KUKA KRL program: f1_Kuka_APT202T02S02.SRC

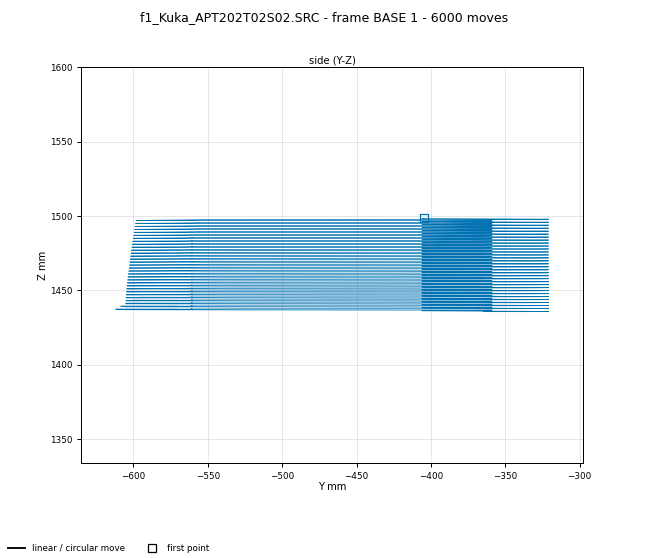
[picture p0: tool path of f1_Kuka_APT202T02S02.SRC in frame BASE 1, 6000 of 6001 moves have a stored position in this frame; points joined in program order, loops and branches not executed]
&ACCESS RVP
&REL 2
&PARAM TEMPLATE = C:\KRC\Roboter\Template\vorgabe
&PARAM EDITMASK = *
DEF f1_Kuka_APT202T02S02()


;FOLD INI;%{PE}%V3.2.0,%MKUKATPBASIS,%CINIT,%VCOMMON,%P
  ;FOLD BAS INI;%{E}%V3.2.0,%MKUKATPBASIS,%CINIT,%VINIT,%P
    GLOBAL INTERRUPT DECL 3 WHEN $STOPMESS==TRUE DO IR_STOPM ( )
    INTERRUPT ON 3
    BAS (#INITMOV,0 )
  ;ENDFOLD (BAS INI)
  ;FOLD USER INI;%{E}%V3.2.0,%MKUKATPUSER,%CINIT,%VINIT,%P
    ;Make your modifications here
  ;ENDFOLD (USER INI)
;ENDFOLD (INI)


;*** Make Null PTP Move
  PTP $pos_act

;*** Auto Load The Correct TOOL Data
  $tool=tool_data[2]

;*** Auto Load The Correct BASE Data
  $base=base_data[1]

  $ADVANCE = 5

;*** Restate Last Velocity
MMPM(30000.0)
SetRPM(8000)
LIN {X -0.079,Y -404.735,Z 1498.391,A 0.000,B 0.000,C 90.000,E1 286.441} C_DIS
LIN {X 0.214,Y -406.099,Z 1498.364,A 0.000,B 0.000,C 90.000,E1 281.535} C_DIS
LIN {X -0.176,Y -406.094,Z 1498.362,A 0.000,B 0.000,C 90.000,E1 281.243} C_DIS
LIN {X -0.097,Y -405.680,Z 1498.333,A 0.000,B 0.000,C 90.000,E1 276.024} C_DIS
LIN {X -0.165,Y -405.058,Z 1498.328,A 0.000,B 0.000,C 90.000,E1 274.992} C_DIS
LIN {X -0.060,Y -403.497,Z 1498.304,A 0.000,B 0.000,C 90.000,E1 270.802} C_DIS
LIN {X -0.092,Y -403.288,Z 1498.302,A 0.000,B 0.000,C 90.000,E1 270.458} C_DIS
LIN {X 0.091,Y -398.931,Z 1498.271,A 0.000,B 0.000,C 90.000,E1 264.837} C_DIS
LIN {X -0.040,Y -393.108,Z 1498.242,A 0.000,B 0.000,C 90.000,E1 259.567} C_DIS
LIN {X -0.079,Y -392.835,Z 1498.240,A 0.000,B 0.000,C 90.000,E1 259.218} C_DIS
LIN {X 0.034,Y -385.993,Z 1498.212,A 0.000,B 0.000,C 90.000,E1 254.212} C_DIS
LIN {X -0.026,Y -385.267,Z 1498.208,A 0.000,B 0.000,C 90.000,E1 253.504} C_DIS
LIN {X -0.004,Y -384.768,Z 1498.206,A 0.000,B 0.000,C 90.000,E1 253.142} C_DIS
LIN {X 0.221,Y -377.973,Z 1498.182,A 0.000,B 0.000,C 90.000,E1 248.773} C_DIS
LIN {X -0.044,Y -376.233,Z 1498.174,A 0.000,B 0.000,C 90.000,E1 247.358} C_DIS
LIN {X 0.057,Y -374.944,Z 1498.170,A 0.000,B 0.000,C 90.000,E1 246.613} C_DIS
LIN {X -0.208,Y -368.417,Z 1498.148,A 0.000,B 0.000,C 90.000,E1 242.615} C_DIS
LIN {X 0.097,Y -366.047,Z 1498.137,A 0.000,B 0.000,C 90.000,E1 240.717} C_DIS
LIN {X 0.004,Y -359.196,Z 1498.115,A 0.000,B 0.000,C 90.000,E1 236.628} C_DIS
LIN {X 0.021,Y -355.842,Z 1498.100,A 0.000,B 0.000,C 90.000,E1 233.989} C_DIS
LIN {X -0.173,Y -348.793,Z 1498.075,A 0.000,B 0.000,C 90.000,E1 229.461} C_DIS
LIN {X -0.097,Y -346.185,Z 1498.062,A 0.000,B 0.000,C 90.000,E1 227.148} C_DIS
LIN {X -0.088,Y -345.065,Z 1498.058,A 0.000,B 0.000,C 90.000,E1 226.377} C_DIS
LIN {X 0.094,Y -338.586,Z 1498.030,A 0.000,B 0.000,C 90.000,E1 221.310} C_DIS
LIN {X 0.094,Y -336.840,Z 1498.019,A 0.000,B 0.000,C 90.000,E1 219.358} C_DIS
LIN {X 0.014,Y -330.861,Z 1497.988,A 0.000,B 0.000,C 90.000,E1 213.865} C_DIS
LIN {X 0.149,Y -329.296,Z 1497.975,A 0.000,B 0.000,C 90.000,E1 211.465} C_DIS
LIN {X -0.154,Y -324.669,Z 1497.942,A 0.000,B 0.000,C 90.000,E1 205.540} C_DIS
LIN {X 0.174,Y -323.837,Z 1497.928,A 0.000,B 0.000,C 90.000,E1 203.078} C_DIS
LIN {X -0.017,Y -321.124,Z 1497.881,A 0.000,B 0.000,C 90.000,E1 194.662} C_DIS
LIN {X 0.138,Y -320.932,Z 1497.877,A 0.000,B 0.000,C 90.000,E1 193.828} C_DIS
LIN {X -0.076,Y -321.562,Z 1497.832,A 0.000,B 0.000,C 90.000,E1 185.796} C_DIS
LIN {X -0.143,Y -324.415,Z 1497.790,A 0.000,B 0.000,C 90.000,E1 178.165} C_DIS
LIN {X -0.141,Y -325.376,Z 1497.783,A 0.000,B 0.000,C 90.000,E1 176.963} C_DIS
LIN {X -0.100,Y -329.112,Z 1497.750,A 0.000,B 0.000,C 90.000,E1 170.971} C_DIS
LIN {X 0.061,Y -334.260,Z 1497.726,A 0.000,B 0.000,C 90.000,E1 166.589} C_DIS
LIN {X 0.067,Y -335.488,Z 1497.719,A 0.000,B 0.000,C 90.000,E1 165.408} C_DIS
LIN {X 0.143,Y -340.932,Z 1497.695,A 0.000,B 0.000,C 90.000,E1 161.094} C_DIS
LIN {X -0.172,Y -342.138,Z 1497.691,A 0.000,B 0.000,C 90.000,E1 160.369} C_DIS
LIN {X -0.058,Y -347.939,Z 1497.667,A 0.000,B 0.000,C 90.000,E1 156.102} C_DIS
LIN {X -0.081,Y -354.259,Z 1497.648,A 0.000,B 0.000,C 90.000,E1 152.666} C_DIS
LIN {X -0.222,Y -361.406,Z 1497.625,A 0.000,B 0.000,C 90.000,E1 148.535} C_DIS
LIN {X 0.128,Y -363.944,Z 1497.618,A 0.000,B 0.000,C 90.000,E1 147.248} C_DIS
LIN {X 0.147,Y -524.568,Z 1497.618,A 0.000,B 0.000,C 90.000,E1 147.248} C_DIS
LIN {X 0.123,Y -527.252,Z 1497.617,A 0.000,B 0.000,C 90.000,E1 147.120} C_DIS
LIN {X 0.098,Y -528.648,Z 1497.617,A 0.000,B 0.000,C 90.000,E1 146.993} C_DIS
LIN {X -0.114,Y -530.734,Z 1497.615,A 0.000,B 0.000,C 90.000,E1 146.755} C_DIS
LIN {X 0.153,Y -533.334,Z 1497.613,A 0.000,B 0.000,C 90.000,E1 146.294} C_DIS
LIN {X 0.143,Y -534.740,Z 1497.611,A 0.000,B 0.000,C 90.000,E1 146.008} C_DIS
LIN {X -0.014,Y -536.490,Z 1497.609,A 0.000,B 0.000,C 90.000,E1 145.595} C_DIS
LIN {X -0.007,Y -538.436,Z 1497.606,A 0.000,B 0.000,C 90.000,E1 145.022} C_DIS
LIN {X -0.295,Y -540.027,Z 1497.603,A 0.000,B 0.000,C 90.000,E1 144.482} C_DIS
LIN {X -0.213,Y -542.835,Z 1497.596,A 0.000,B 0.000,C 90.000,E1 143.336} C_DIS
LIN {X -0.052,Y -545.857,Z 1497.588,A 0.000,B 0.000,C 90.000,E1 141.904} C_DIS
LIN {X 0.073,Y -548.299,Z 1497.581,A 0.000,B 0.000,C 90.000,E1 140.481} C_DIS
LIN {X -0.110,Y -550.441,Z 1497.573,A 0.000,B 0.000,C 90.000,E1 139.094} C_DIS
LIN {X 0.036,Y -551.981,Z 1497.567,A 0.000,B 0.000,C 90.000,E1 137.957} C_DIS
LIN {X -0.256,Y -553.028,Z 1497.562,A 0.000,B 0.000,C 90.000,E1 137.148} C_DIS
LIN {X -0.045,Y -554.642,Z 1497.554,A 0.000,B 0.000,C 90.000,E1 135.729} C_DIS
LIN {X 0.139,Y -555.726,Z 1497.548,A 0.000,B 0.000,C 90.000,E1 134.595} C_DIS
LIN {X -0.006,Y -556.926,Z 1497.540,A 0.000,B 0.000,C 90.000,E1 133.218} C_DIS
LIN {X -0.108,Y -557.910,Z 1497.532,A 0.000,B 0.000,C 90.000,E1 131.838} C_DIS
LIN {X -0.191,Y -558.747,Z 1497.525,A 0.000,B 0.000,C 90.000,E1 130.458} C_DIS
LIN {X 0.161,Y -559.408,Z 1497.517,A 0.000,B 0.000,C 90.000,E1 129.036} C_DIS
LIN {X 0.170,Y -559.997,Z 1497.509,A 0.000,B 0.000,C 90.000,E1 127.649} C_DIS
LIN {X -0.243,Y -560.290,Z 1497.503,A 0.000,B 0.000,C 90.000,E1 126.583} C_DIS
LIN {X -0.099,Y -560.494,Z 1497.495,A 0.000,B 0.000,C 90.000,E1 125.185} C_DIS
LIN {X 0.181,Y -560.465,Z 1497.491,A 0.000,B 0.000,C 90.000,E1 124.326} C_DIS
LIN {X 0.011,Y -560.350,Z 1497.483,A 0.000,B 0.000,C 90.000,E1 122.959} C_DIS
LIN {X 0.188,Y -560.363,Z 1497.472,A 0.000,B 0.000,C 90.000,E1 121.003} C_DIS
LIN {X 0.280,Y -560.586,Z 1497.463,A 0.000,B 0.000,C 90.000,E1 119.333} C_DIS
LIN {X -0.170,Y -560.853,Z 1497.454,A 0.000,B 0.000,C 90.000,E1 117.719} C_DIS
LIN {X 0.244,Y -561.212,Z 1497.442,A 0.000,B 0.000,C 90.000,E1 115.463} C_DIS
LIN {X 0.063,Y -561.585,Z 1497.432,A 0.000,B 0.000,C 90.000,E1 113.823} C_DIS
LIN {X 0.068,Y -561.889,Z 1497.426,A 0.000,B 0.000,C 90.000,E1 112.717} C_DIS
LIN {X -0.004,Y -562.293,Z 1497.416,A 0.000,B 0.000,C 90.000,E1 110.791} C_DIS
LIN {X -0.075,Y -562.700,Z 1497.406,A 0.000,B 0.000,C 90.000,E1 109.141} C_DIS
LIN {X 0.211,Y -563.076,Z 1497.397,A 0.000,B 0.000,C 90.000,E1 107.457} C_DIS
LIN {X -0.196,Y -563.524,Z 1497.388,A 0.000,B 0.000,C 90.000,E1 105.843} C_DIS
LIN {X 0.101,Y -564.102,Z 1497.377,A 0.000,B 0.000,C 90.000,E1 103.883} C_DIS
LIN {X -0.237,Y -564.827,Z 1497.365,A 0.000,B 0.000,C 90.000,E1 101.715} C_DIS
LIN {X 0.046,Y -565.361,Z 1497.357,A 0.000,B 0.000,C 90.000,E1 100.310} C_DIS
LIN {X 0.066,Y -565.901,Z 1497.351,A 0.000,B 0.000,C 90.000,E1 99.208} C_DIS
LIN {X 0.262,Y -566.469,Z 1497.344,A 0.000,B 0.000,C 90.000,E1 97.814} C_DIS
LIN {X -0.210,Y -567.729,Z 1497.330,A 0.000,B 0.000,C 90.000,E1 95.391} C_DIS
LIN {X -0.124,Y -568.501,Z 1497.322,A 0.000,B 0.000,C 90.000,E1 94.012} C_DIS
LIN {X -0.182,Y -569.180,Z 1497.316,A 0.000,B 0.000,C 90.000,E1 92.922} C_DIS
LIN {X -0.104,Y -570.043,Z 1497.309,A 0.000,B 0.000,C 90.000,E1 91.547} C_DIS
LIN {X 0.111,Y -571.078,Z 1497.299,A 0.000,B 0.000,C 90.000,E1 89.885} C_DIS
LIN {X -0.069,Y -572.412,Z 1497.289,A 0.000,B 0.000,C 90.000,E1 87.993} C_DIS
LIN {X 0.076,Y -573.269,Z 1497.281,A 0.000,B 0.000,C 90.000,E1 86.617} C_DIS
LIN {X -0.165,Y -574.340,Z 1497.272,A 0.000,B 0.000,C 90.000,E1 85.008} C_DIS
LIN {X 0.241,Y -575.491,Z 1497.263,A 0.000,B 0.000,C 90.000,E1 83.337} C_DIS
LIN {X -0.065,Y -577.062,Z 1497.251,A 0.000,B 0.000,C 90.000,E1 81.197} C_DIS
LIN {X 0.101,Y -578.510,Z 1497.241,A 0.000,B 0.000,C 90.000,E1 79.285} C_DIS
LIN {X -0.055,Y -580.003,Z 1497.230,A 0.000,B 0.000,C 90.000,E1 77.409} C_DIS
LIN {X 0.301,Y -581.227,Z 1497.221,A 0.000,B 0.000,C 90.000,E1 75.755} C_DIS
LIN {X 0.121,Y -582.355,Z 1497.212,A 0.000,B 0.000,C 90.000,E1 74.157} C_DIS
LIN {X 0.116,Y -583.325,Z 1497.203,A 0.000,B 0.000,C 90.000,E1 72.543} C_DIS
LIN {X -0.097,Y -584.064,Z 1497.196,A 0.000,B 0.000,C 90.000,E1 71.221} C_DIS
LIN {X 0.301,Y -584.970,Z 1497.187,A 0.000,B 0.000,C 90.000,E1 69.571} C_DIS
LIN {X -0.302,Y -586.230,Z 1497.175,A 0.000,B 0.000,C 90.000,E1 67.486} C_DIS
LIN {X -0.310,Y -587.282,Z 1497.164,A 0.000,B 0.000,C 90.000,E1 65.613} C_DIS
LIN {X -0.052,Y -588.468,Z 1497.154,A 0.000,B 0.000,C 90.000,E1 63.717} C_DIS
LIN {X -0.032,Y -589.765,Z 1497.144,A 0.000,B 0.000,C 90.000,E1 61.847} C_DIS
LIN {X -0.108,Y -590.882,Z 1497.135,A 0.000,B 0.000,C 90.000,E1 60.255} C_DIS
LIN {X -0.260,Y -592.270,Z 1497.124,A 0.000,B 0.000,C 90.000,E1 58.408} C_DIS
LIN {X 0.022,Y -593.566,Z 1497.116,A 0.000,B 0.000,C 90.000,E1 56.786} C_DIS
LIN {X -0.056,Y -594.604,Z 1497.108,A 0.000,B 0.000,C 90.000,E1 55.468} C_DIS
LIN {X 0.106,Y -595.700,Z 1497.099,A 0.000,B 0.000,C 90.000,E1 53.863} C_DIS
LIN {X 0.310,Y -596.099,Z 1497.095,A 0.000,B 0.000,C 90.000,E1 53.050} C_DIS
LIN {X -0.227,Y -596.917,Z 1497.085,A 0.000,B 0.000,C 90.000,E1 51.251} C_DIS
LIN {X -0.229,Y -597.429,Z 1497.079,A 0.000,B 0.000,C 90.000,E1 50.194} C_DIS
LIN {X 0.003,Y -597.888,Z 1497.074,A 0.000,B 0.000,C 90.000,E1 49.380} C_DIS
LIN {X 0.014,Y -598.188,Z 1497.068,A 0.000,B 0.000,C 90.000,E1 48.324} C_DIS
LIN {X 0.020,Y -598.255,Z 1497.063,A 0.000,B 0.000,C 90.000,E1 47.268} C_DIS
LIN {X 0.212,Y -598.199,Z 1497.058,A 0.000,B 0.000,C 90.000,E1 46.458} C_DIS
LIN {X -0.024,Y -597.979,Z 1497.051,A 0.000,B 0.000,C 90.000,E1 45.162} C_DIS
LIN {X -0.043,Y -597.462,Z 1497.045,A 0.000,B 0.000,C 90.000,E1 44.109} C_DIS
LIN {X 0.144,Y -596.988,Z 1497.041,A 0.000,B 0.000,C 90.000,E1 43.299} C_DIS
LIN {X -0.090,Y -595.920,Z 1497.033,A 0.000,B 0.000,C 90.000,E1 42.000} C_DIS
LIN {X -0.324,Y -595.174,Z 1497.029,A 0.000,B 0.000,C 90.000,E1 41.229} C_DIS
LIN {X -0.132,Y -593.586,Z 1497.022,A 0.000,B 0.000,C 90.000,E1 39.886} C_DIS
LIN {X 0.062,Y -592.515,Z 1497.017,A 0.000,B 0.000,C 90.000,E1 39.072} C_DIS
LIN {X 0.200,Y -590.340,Z 1497.010,A 0.000,B 0.000,C 90.000,E1 37.729} C_DIS
LIN {X 0.198,Y -588.199,Z 1497.004,A 0.000,B 0.000,C 90.000,E1 36.664} C_DIS
LIN {X -0.025,Y -586.372,Z 1496.999,A 0.000,B 0.000,C 90.000,E1 35.884} C_DIS
LIN {X -0.268,Y -584.413,Z 1496.995,A 0.000,B 0.000,C 90.000,E1 35.105} C_DIS
LIN {X -0.050,Y -582.104,Z 1496.990,A 0.000,B 0.000,C 90.000,E1 34.278} C_DIS
LIN {X -0.175,Y -578.675,Z 1496.984,A 0.000,B 0.000,C 90.000,E1 33.214} C_DIS
LIN {X -0.336,Y -575.589,Z 1496.980,A 0.000,B 0.000,C 90.000,E1 32.418} C_DIS
LIN {X -0.050,Y -573.175,Z 1496.977,A 0.000,B 0.000,C 90.000,E1 31.848} C_DIS
LIN {X -0.304,Y -570.965,Z 1496.975,A 0.000,B 0.000,C 90.000,E1 31.465} C_DIS
LIN {X 0.218,Y -568.308,Z 1496.972,A 0.000,B 0.000,C 90.000,E1 31.003} C_DIS
LIN {X 0.039,Y -566.164,Z 1496.971,A 0.000,B 0.000,C 90.000,E1 30.747} C_DIS
LIN {X 0.235,Y -564.885,Z 1496.970,A 0.000,B 0.000,C 90.000,E1 30.590} C_DIS
LIN {X 0.084,Y -562.667,Z 1496.969,A 0.000,B 0.000,C 90.000,E1 30.413} C_DIS
LIN {X -0.176,Y -560.913,Z 1496.969,A 0.000,B 0.000,C 90.000,E1 30.335} C_DIS
LIN {X 0.114,Y -559.281,Z 1496.968,A 0.000,B 0.000,C 90.000,E1 30.256} C_DIS
LIN {X 0.055,Y -390.789,Z 1496.968,A 0.000,B 0.000,C 90.000,E1 30.256} C_DIS
LIN {X -0.100,Y -383.744,Z 1496.942,A 0.000,B 0.000,C 90.000,E1 25.591} C_DIS
LIN {X 0.062,Y -382.915,Z 1496.938,A 0.000,B 0.000,C 90.000,E1 24.847} C_DIS
LIN {X 0.168,Y -376.206,Z 1496.912,A 0.000,B 0.000,C 90.000,E1 20.120} C_DIS
LIN {X 0.036,Y -373.711,Z 1496.898,A 0.000,B 0.000,C 90.000,E1 17.583} C_DIS
LIN {X 0.172,Y -368.106,Z 1496.869,A 0.000,B 0.000,C 90.000,E1 12.411} C_DIS
LIN {X -0.022,Y -366.430,Z 1496.855,A 0.000,B 0.000,C 90.000,E1 9.849} C_DIS
LIN {X -0.084,Y -361.753,Z 1496.822,A 0.000,B 0.000,C 90.000,E1 3.898} C_DIS
LIN {X 0.163,Y -360.877,Z 1496.801,A 0.000,B 0.000,C 90.000,E1 0.115} C_DIS
LIN {X -0.053,Y -359.426,Z 1496.770,A 0.000,B 0.000,C 90.000,E1 354.546} C_DIS
LIN {X 0.070,Y -358.890,Z 1496.759,A 0.000,B 0.000,C 90.000,E1 352.648} C_DIS
LIN {X -0.020,Y -359.563,Z 1496.726,A 0.000,B 0.000,C 90.000,E1 346.645} C_DIS
LIN {X 0.001,Y -361.801,Z 1496.684,A 0.000,B 0.000,C 90.000,E1 339.135} C_DIS
LIN {X -0.154,Y -362.053,Z 1496.680,A 0.000,B 0.000,C 90.000,E1 338.411} C_DIS
LIN {X 0.189,Y -365.980,Z 1496.643,A 0.000,B 0.000,C 90.000,E1 331.641} C_DIS
LIN {X 0.029,Y -366.387,Z 1496.639,A 0.000,B 0.000,C 90.000,E1 330.923} C_DIS
LIN {X -0.031,Y -371.355,Z 1496.604,A 0.000,B 0.000,C 90.000,E1 324.642} C_DIS
LIN {X -0.043,Y -371.766,Z 1496.602,A 0.000,B 0.000,C 90.000,E1 324.276} C_DIS
LIN {X 0.013,Y -377.358,Z 1496.567,A 0.000,B 0.000,C 90.000,E1 318.038} C_DIS
LIN {X 0.012,Y -378.235,Z 1496.563,A 0.000,B 0.000,C 90.000,E1 317.310} C_DIS
LIN {X 0.002,Y -383.940,Z 1496.531,A 0.000,B 0.000,C 90.000,E1 311.515} C_DIS
LIN {X 0.088,Y -384.893,Z 1496.527,A 0.000,B 0.000,C 90.000,E1 310.782} C_DIS
LIN {X 0.262,Y -390.610,Z 1496.495,A 0.000,B 0.000,C 90.000,E1 305.025} C_DIS
LIN {X 0.106,Y -391.104,Z 1496.493,A 0.000,B 0.000,C 90.000,E1 304.692} C_DIS
LIN {X 0.022,Y -391.648,Z 1496.489,A 0.000,B 0.000,C 90.000,E1 303.992} C_DIS
LIN {X -0.080,Y -396.825,Z 1496.459,A 0.000,B 0.000,C 90.000,E1 298.693} C_DIS
LIN {X -0.210,Y -397.120,Z 1496.457,A 0.000,B 0.000,C 90.000,E1 298.359} C_DIS
LIN {X -0.055,Y -401.597,Z 1496.426,A 0.000,B 0.000,C 90.000,E1 292.717} C_DIS
LIN {X 0.222,Y -404.659,Z 1496.395,A 0.000,B 0.000,C 90.000,E1 287.094} C_DIS
LIN {X -0.079,Y -404.735,Z 1496.391,A 0.000,B 0.000,C 90.000,E1 286.441} C_DIS
LIN {X 0.214,Y -406.099,Z 1496.364,A 0.000,B 0.000,C 90.000,E1 281.535} C_DIS
LIN {X -0.176,Y -406.094,Z 1496.362,A 0.000,B 0.000,C 90.000,E1 281.243} C_DIS
LIN {X -0.097,Y -405.680,Z 1496.333,A 0.000,B 0.000,C 90.000,E1 276.024} C_DIS
LIN {X -0.165,Y -405.058,Z 1496.328,A 0.000,B 0.000,C 90.000,E1 274.992} C_DIS
LIN {X -0.060,Y -403.497,Z 1496.304,A 0.000,B 0.000,C 90.000,E1 270.802} C_DIS
LIN {X -0.092,Y -403.288,Z 1496.302,A 0.000,B 0.000,C 90.000,E1 270.458} C_DIS
LIN {X 0.091,Y -398.931,Z 1496.271,A 0.000,B 0.000,C 90.000,E1 264.837} C_DIS
LIN {X -0.040,Y -393.108,Z 1496.242,A 0.000,B 0.000,C 90.000,E1 259.567} C_DIS
LIN {X -0.079,Y -392.835,Z 1496.240,A 0.000,B 0.000,C 90.000,E1 259.218} C_DIS
LIN {X 0.034,Y -385.993,Z 1496.212,A 0.000,B 0.000,C 90.000,E1 254.212} C_DIS
LIN {X -0.026,Y -385.267,Z 1496.208,A 0.000,B 0.000,C 90.000,E1 253.504} C_DIS
LIN {X -0.004,Y -384.768,Z 1496.206,A 0.000,B 0.000,C 90.000,E1 253.142} C_DIS
LIN {X 0.221,Y -377.973,Z 1496.182,A 0.000,B 0.000,C 90.000,E1 248.773} C_DIS
LIN {X -0.044,Y -376.233,Z 1496.174,A 0.000,B 0.000,C 90.000,E1 247.358} C_DIS
LIN {X 0.057,Y -374.944,Z 1496.170,A 0.000,B 0.000,C 90.000,E1 246.613} C_DIS
LIN {X -0.208,Y -368.417,Z 1496.148,A 0.000,B 0.000,C 90.000,E1 242.615} C_DIS
LIN {X 0.097,Y -366.047,Z 1496.137,A 0.000,B 0.000,C 90.000,E1 240.717} C_DIS
LIN {X 0.004,Y -359.196,Z 1496.115,A 0.000,B 0.000,C 90.000,E1 236.628} C_DIS
LIN {X 0.021,Y -355.842,Z 1496.100,A 0.000,B 0.000,C 90.000,E1 233.989} C_DIS
LIN {X -0.173,Y -348.793,Z 1496.075,A 0.000,B 0.000,C 90.000,E1 229.461} C_DIS
LIN {X -0.097,Y -346.185,Z 1496.062,A 0.000,B 0.000,C 90.000,E1 227.148} C_DIS
LIN {X -0.088,Y -345.065,Z 1496.058,A 0.000,B 0.000,C 90.000,E1 226.377} C_DIS
LIN {X 0.094,Y -338.586,Z 1496.030,A 0.000,B 0.000,C 90.000,E1 221.310} C_DIS
LIN {X 0.094,Y -336.840,Z 1496.019,A 0.000,B 0.000,C 90.000,E1 219.358} C_DIS
LIN {X 0.014,Y -330.861,Z 1495.988,A 0.000,B 0.000,C 90.000,E1 213.865} C_DIS
LIN {X 0.149,Y -329.296,Z 1495.975,A 0.000,B 0.000,C 90.000,E1 211.465} C_DIS
LIN {X -0.154,Y -324.669,Z 1495.942,A 0.000,B 0.000,C 90.000,E1 205.540} C_DIS
LIN {X 0.174,Y -323.837,Z 1495.928,A 0.000,B 0.000,C 90.000,E1 203.078} C_DIS
LIN {X -0.017,Y -321.124,Z 1495.881,A 0.000,B 0.000,C 90.000,E1 194.662} C_DIS
LIN {X 0.138,Y -320.932,Z 1495.877,A 0.000,B 0.000,C 90.000,E1 193.828} C_DIS
LIN {X -0.076,Y -321.562,Z 1495.832,A 0.000,B 0.000,C 90.000,E1 185.796} C_DIS
LIN {X -0.143,Y -324.415,Z 1495.790,A 0.000,B 0.000,C 90.000,E1 178.165} C_DIS
LIN {X -0.141,Y -325.376,Z 1495.783,A 0.000,B 0.000,C 90.000,E1 176.963} C_DIS
LIN {X -0.100,Y -329.112,Z 1495.750,A 0.000,B 0.000,C 90.000,E1 170.971} C_DIS
LIN {X 0.061,Y -334.260,Z 1495.726,A 0.000,B 0.000,C 90.000,E1 166.589} C_DIS
LIN {X 0.067,Y -335.488,Z 1495.719,A 0.000,B 0.000,C 90.000,E1 165.408} C_DIS
LIN {X 0.143,Y -340.932,Z 1495.695,A 0.000,B 0.000,C 90.000,E1 161.094} C_DIS
LIN {X -0.172,Y -342.138,Z 1495.691,A 0.000,B 0.000,C 90.000,E1 160.369} C_DIS
LIN {X -0.058,Y -347.939,Z 1495.667,A 0.000,B 0.000,C 90.000,E1 156.102} C_DIS
LIN {X -0.081,Y -354.259,Z 1495.648,A 0.000,B 0.000,C 90.000,E1 152.666} C_DIS
LIN {X -0.222,Y -361.406,Z 1495.625,A 0.000,B 0.000,C 90.000,E1 148.535} C_DIS
LIN {X -0.211,Y -362.490,Z 1495.622,A 0.000,B 0.000,C 90.000,E1 147.995} C_DIS
LIN {X 0.110,Y -522.437,Z 1495.622,A 0.000,B 0.000,C 90.000,E1 147.946} C_DIS
LIN {X -0.131,Y -524.949,Z 1495.621,A 0.000,B 0.000,C 90.000,E1 147.867} C_DIS
LIN {X 0.102,Y -526.192,Z 1495.621,A 0.000,B 0.000,C 90.000,E1 147.740} C_DIS
LIN {X 0.059,Y -528.355,Z 1495.620,A 0.000,B 0.000,C 90.000,E1 147.502} C_DIS
LIN {X -0.243,Y -530.287,Z 1495.618,A 0.000,B 0.000,C 90.000,E1 147.248} C_DIS
LIN {X 0.022,Y -532.672,Z 1495.616,A 0.000,B 0.000,C 90.000,E1 146.786} C_DIS
LIN {X -0.147,Y -534.604,Z 1495.613,A 0.000,B 0.000,C 90.000,E1 146.373} C_DIS
LIN {X -0.154,Y -535.744,Z 1495.612,A 0.000,B 0.000,C 90.000,E1 146.087} C_DIS
LIN {X -0.156,Y -537.582,Z 1495.608,A 0.000,B 0.000,C 90.000,E1 145.515} C_DIS
LIN {X 0.003,Y -539.990,Z 1495.604,A 0.000,B 0.000,C 90.000,E1 144.642} C_DIS
LIN {X 0.057,Y -542.139,Z 1495.599,A 0.000,B 0.000,C 90.000,E1 143.783} C_DIS
LIN {X 0.137,Y -544.076,Z 1495.594,A 0.000,B 0.000,C 90.000,E1 142.924} C_DIS
LIN {X -0.192,Y -545.882,Z 1495.589,A 0.000,B 0.000,C 90.000,E1 142.110} C_DIS
LIN {X -0.029,Y -547.881,Z 1495.583,A 0.000,B 0.000,C 90.000,E1 140.964} C_DIS
LIN {X 0.082,Y -549.671,Z 1495.577,A 0.000,B 0.000,C 90.000,E1 139.828} C_DIS
LIN {X 0.224,Y -551.300,Z 1495.571,A 0.000,B 0.000,C 90.000,E1 138.690} C_DIS
LIN {X -0.021,Y -552.782,Z 1495.564,A 0.000,B 0.000,C 90.000,E1 137.595} C_DIS
LIN {X 0.244,Y -554.722,Z 1495.555,A 0.000,B 0.000,C 90.000,E1 135.891} C_DIS
LIN {X 0.035,Y -555.819,Z 1495.549,A 0.000,B 0.000,C 90.000,E1 134.798} C_DIS
LIN {X -0.095,Y -557.046,Z 1495.541,A 0.000,B 0.000,C 90.000,E1 133.419} C_DIS
LIN {X 0.189,Y -558.017,Z 1495.533,A 0.000,B 0.000,C 90.000,E1 132.000} C_DIS
LIN {X 0.030,Y -558.685,Z 1495.527,A 0.000,B 0.000,C 90.000,E1 130.906} C_DIS
LIN {X -0.062,Y -559.255,Z 1495.521,A 0.000,B 0.000,C 90.000,E1 129.806} C_DIS
LIN {X 0.302,Y -559.823,Z 1495.513,A 0.000,B 0.000,C 90.000,E1 128.382} C_DIS
LIN {X -0.208,Y -560.128,Z 1495.509,A 0.000,B 0.000,C 90.000,E1 127.604} C_DIS
LIN {X 0.076,Y -560.338,Z 1495.504,A 0.000,B 0.000,C 90.000,E1 126.744} C_DIS
LIN {X -0.232,Y -560.549,Z 1495.497,A 0.000,B 0.000,C 90.000,E1 125.391} C_DIS
LIN {X -0.174,Y -560.489,Z 1495.490,A 0.000,B 0.000,C 90.000,E1 124.278} C_DIS
LIN {X -0.032,Y -560.362,Z 1495.483,A 0.000,B 0.000,C 90.000,E1 122.880} C_DIS
LIN {X 0.139,Y -560.395,Z 1495.472,A 0.000,B 0.000,C 90.000,E1 120.924} C_DIS
LIN {X -0.047,Y -560.625,Z 1495.463,A 0.000,B 0.000,C 90.000,E1 119.283} C_DIS
LIN {X 0.068,Y -560.940,Z 1495.452,A 0.000,B 0.000,C 90.000,E1 117.334} C_DIS
LIN {X -0.265,Y -561.309,Z 1495.440,A 0.000,B 0.000,C 90.000,E1 115.155} C_DIS
LIN {X -0.126,Y -561.830,Z 1495.429,A 0.000,B 0.000,C 90.000,E1 113.206} C_DIS
LIN {X 0.003,Y -562.154,Z 1495.420,A 0.000,B 0.000,C 90.000,E1 111.535} C_DIS
LIN {X -0.062,Y -562.534,Z 1495.411,A 0.000,B 0.000,C 90.000,E1 109.885} C_DIS
LIN {X -0.126,Y -562.961,Z 1495.401,A 0.000,B 0.000,C 90.000,E1 108.236} C_DIS
LIN {X -0.228,Y -563.464,Z 1495.391,A 0.000,B 0.000,C 90.000,E1 106.315} C_DIS
LIN {X 0.224,Y -564.103,Z 1495.378,A 0.000,B 0.000,C 90.000,E1 104.064} C_DIS
LIN {X 0.232,Y -564.617,Z 1495.369,A 0.000,B 0.000,C 90.000,E1 102.411} C_DIS
LIN {X 0.013,Y -565.272,Z 1495.360,A 0.000,B 0.000,C 90.000,E1 100.782} C_DIS
LIN {X -0.182,Y -566.027,Z 1495.351,A 0.000,B 0.000,C 90.000,E1 99.151} C_DIS
LIN {X 0.018,Y -566.588,Z 1495.343,A 0.000,B 0.000,C 90.000,E1 97.757} C_DIS
LIN {X -0.045,Y -567.731,Z 1495.331,A 0.000,B 0.000,C 90.000,E1 95.568} C_DIS
LIN {X 0.209,Y -568.649,Z 1495.322,A 0.000,B 0.000,C 90.000,E1 93.898} C_DIS
LIN {X 0.154,Y -569.353,Z 1495.316,A 0.000,B 0.000,C 90.000,E1 92.808} C_DIS
LIN {X 0.237,Y -570.216,Z 1495.308,A 0.000,B 0.000,C 90.000,E1 91.432} C_DIS
LIN {X -0.247,Y -571.113,Z 1495.301,A 0.000,B 0.000,C 90.000,E1 90.115} C_DIS
LIN {X -0.009,Y -572.252,Z 1495.292,A 0.000,B 0.000,C 90.000,E1 88.453} C_DIS
LIN {X 0.124,Y -573.175,Z 1495.284,A 0.000,B 0.000,C 90.000,E1 87.078} C_DIS
LIN {X -0.125,Y -574.223,Z 1495.275,A 0.000,B 0.000,C 90.000,E1 85.469} C_DIS
LIN {X 0.273,Y -575.363,Z 1495.266,A 0.000,B 0.000,C 90.000,E1 83.799} C_DIS
LIN {X -0.245,Y -576.726,Z 1495.255,A 0.000,B 0.000,C 90.000,E1 81.951} C_DIS
LIN {X -0.295,Y -577.948,Z 1495.246,A 0.000,B 0.000,C 90.000,E1 80.330} C_DIS
LIN {X 0.006,Y -578.821,Z 1495.240,A 0.000,B 0.000,C 90.000,E1 79.218} C_DIS
LIN {X 0.088,Y -580.090,Z 1495.231,A 0.000,B 0.000,C 90.000,E1 77.589} C_DIS
LIN {X 0.214,Y -581.171,Z 1495.224,A 0.000,B 0.000,C 90.000,E1 76.228} C_DIS
LIN {X -0.192,Y -582.130,Z 1495.216,A 0.000,B 0.000,C 90.000,E1 74.921} C_DIS
LIN {X -0.022,Y -583.002,Z 1495.209,A 0.000,B 0.000,C 90.000,E1 73.559} C_DIS
LIN {X -0.236,Y -583.767,Z 1495.201,A 0.000,B 0.000,C 90.000,E1 72.236} C_DIS
LIN {X -0.101,Y -584.374,Z 1495.195,A 0.000,B 0.000,C 90.000,E1 71.148} C_DIS
LIN {X 0.109,Y -585.258,Z 1495.186,A 0.000,B 0.000,C 90.000,E1 69.518} C_DIS
LIN {X 0.272,Y -586.506,Z 1495.174,A 0.000,B 0.000,C 90.000,E1 67.358} C_DIS
LIN {X 0.274,Y -587.593,Z 1495.164,A 0.000,B 0.000,C 90.000,E1 65.485} C_DIS
LIN {X 0.015,Y -588.761,Z 1495.154,A 0.000,B 0.000,C 90.000,E1 63.640} C_DIS
LIN {X 0.050,Y -590.034,Z 1495.143,A 0.000,B 0.000,C 90.000,E1 61.769} C_DIS
LIN {X -0.307,Y -591.165,Z 1495.134,A 0.000,B 0.000,C 90.000,E1 60.205} C_DIS
LIN {X -0.152,Y -592.596,Z 1495.124,A 0.000,B 0.000,C 90.000,E1 58.329} C_DIS
LIN {X 0.142,Y -593.861,Z 1495.115,A 0.000,B 0.000,C 90.000,E1 56.707} C_DIS
LIN {X 0.074,Y -594.943,Z 1495.108,A 0.000,B 0.000,C 90.000,E1 55.388} C_DIS
LIN {X 0.247,Y -596.049,Z 1495.099,A 0.000,B 0.000,C 90.000,E1 53.783} C_DIS
LIN {X -0.148,Y -596.553,Z 1495.093,A 0.000,B 0.000,C 90.000,E1 52.763} C_DIS
LIN {X -0.067,Y -597.271,Z 1495.084,A 0.000,B 0.000,C 90.000,E1 51.170} C_DIS
LIN {X -0.064,Y -597.787,Z 1495.078,A 0.000,B 0.000,C 90.000,E1 50.114} C_DIS
LIN {X 0.174,Y -598.232,Z 1495.074,A 0.000,B 0.000,C 90.000,E1 49.299} C_DIS
LIN {X 0.190,Y -598.511,Z 1495.068,A 0.000,B 0.000,C 90.000,E1 48.243} C_DIS
LIN {X -0.237,Y -598.581,Z 1495.062,A 0.000,B 0.000,C 90.000,E1 47.229} C_DIS
LIN {X -0.036,Y -598.513,Z 1495.058,A 0.000,B 0.000,C 90.000,E1 46.419} C_DIS
LIN {X 0.168,Y -598.285,Z 1495.051,A 0.000,B 0.000,C 90.000,E1 45.081} C_DIS
LIN {X 0.153,Y -597.773,Z 1495.045,A 0.000,B 0.000,C 90.000,E1 44.028} C_DIS
LIN {X -0.067,Y -597.302,Z 1495.040,A 0.000,B 0.000,C 90.000,E1 43.257} C_DIS
LIN {X 0.113,Y -596.230,Z 1495.033,A 0.000,B 0.000,C 90.000,E1 41.919} C_DIS
LIN {X -0.120,Y -595.446,Z 1495.029,A 0.000,B 0.000,C 90.000,E1 41.148} C_DIS
LIN {X -0.144,Y -594.237,Z 1495.023,A 0.000,B 0.000,C 90.000,E1 40.092} C_DIS
LIN {X -0.189,Y -592.764,Z 1495.017,A 0.000,B 0.000,C 90.000,E1 39.036} C_DIS
LIN {X -0.162,Y -591.058,Z 1495.011,A 0.000,B 0.000,C 90.000,E1 37.971} C_DIS
LIN {X 0.206,Y -589.018,Z 1495.005,A 0.000,B 0.000,C 90.000,E1 36.870} C_DIS
LIN {X -0.211,Y -587.928,Z 1495.002,A 0.000,B 0.000,C 90.000,E1 36.377} C_DIS
LIN {X -0.245,Y -585.364,Z 1494.996,A 0.000,B 0.000,C 90.000,E1 35.311} C_DIS
LIN {X -0.017,Y -583.180,Z 1494.992,A 0.000,B 0.000,C 90.000,E1 34.485} C_DIS
LIN {X -0.127,Y -579.850,Z 1494.986,A 0.000,B 0.000,C 90.000,E1 33.420} C_DIS
LIN {X -0.121,Y -577.955,Z 1494.983,A 0.000,B 0.000,C 90.000,E1 32.880} C_DIS
LIN {X 0.021,Y -574.761,Z 1494.978,A 0.000,B 0.000,C 90.000,E1 32.054} C_DIS
LIN {X -0.091,Y -571.728,Z 1494.974,A 0.000,B 0.000,C 90.000,E1 31.386} C_DIS
LIN {X -0.143,Y -568.756,Z 1494.971,A 0.000,B 0.000,C 90.000,E1 30.846} C_DIS
LIN {X 0.077,Y -565.975,Z 1494.969,A 0.000,B 0.000,C 90.000,E1 30.413} C_DIS
LIN {X 0.178,Y -563.742,Z 1494.968,A 0.000,B 0.000,C 90.000,E1 30.129} C_DIS
LIN {X 0.081,Y -562.439,Z 1494.967,A 0.000,B 0.000,C 90.000,E1 30.001} C_DIS
LIN {X -0.016,Y -559.895,Z 1494.966,A 0.000,B 0.000,C 90.000,E1 29.795} C_DIS
LIN {X 0.159,Y -557.890,Z 1494.965,A 0.000,B 0.000,C 90.000,E1 29.667} C_DIS
LIN {X -0.147,Y -556.512,Z 1494.965,A 0.000,B 0.000,C 90.000,E1 29.667} C_DIS
LIN {X -0.127,Y -389.695,Z 1494.965,A 0.000,B 0.000,C 90.000,E1 29.667} C_DIS
LIN {X 0.087,Y -383.035,Z 1494.939,A 0.000,B 0.000,C 90.000,E1 24.951} C_DIS
LIN {X -0.105,Y -381.915,Z 1494.935,A 0.000,B 0.000,C 90.000,E1 24.259} C_DIS
LIN {X 0.018,Y -375.527,Z 1494.909,A 0.000,B 0.000,C 90.000,E1 19.523} C_DIS
LIN {X 0.012,Y -373.428,Z 1494.896,A 0.000,B 0.000,C 90.000,E1 17.330} C_DIS
LIN {X -0.054,Y -367.906,Z 1494.868,A 0.000,B 0.000,C 90.000,E1 12.187} C_DIS
LIN {X -0.034,Y -366.504,Z 1494.855,A 0.000,B 0.000,C 90.000,E1 9.962} C_DIS
LIN {X -0.099,Y -361.803,Z 1494.822,A 0.000,B 0.000,C 90.000,E1 4.012} C_DIS
LIN {X 0.147,Y -360.903,Z 1494.802,A 0.000,B 0.000,C 90.000,E1 0.229} C_DIS
LIN {X -0.053,Y -359.426,Z 1494.770,A 0.000,B 0.000,C 90.000,E1 354.546} C_DIS
LIN {X 0.070,Y -358.890,Z 1494.759,A 0.000,B 0.000,C 90.000,E1 352.648} C_DIS
LIN {X -0.020,Y -359.563,Z 1494.726,A 0.000,B 0.000,C 90.000,E1 346.645} C_DIS
LIN {X 0.001,Y -361.801,Z 1494.684,A 0.000,B 0.000,C 90.000,E1 339.135} C_DIS
LIN {X -0.154,Y -362.053,Z 1494.680,A 0.000,B 0.000,C 90.000,E1 338.411} C_DIS
LIN {X 0.189,Y -365.980,Z 1494.643,A 0.000,B 0.000,C 90.000,E1 331.641} C_DIS
LIN {X 0.029,Y -366.387,Z 1494.639,A 0.000,B 0.000,C 90.000,E1 330.923} C_DIS
LIN {X -0.031,Y -371.355,Z 1494.604,A 0.000,B 0.000,C 90.000,E1 324.642} C_DIS
LIN {X -0.043,Y -371.766,Z 1494.602,A 0.000,B 0.000,C 90.000,E1 324.276} C_DIS
LIN {X 0.013,Y -377.358,Z 1494.567,A 0.000,B 0.000,C 90.000,E1 318.038} C_DIS
LIN {X 0.012,Y -378.235,Z 1494.563,A 0.000,B 0.000,C 90.000,E1 317.310} C_DIS
LIN {X 0.002,Y -383.940,Z 1494.531,A 0.000,B 0.000,C 90.000,E1 311.515} C_DIS
LIN {X 0.088,Y -384.893,Z 1494.527,A 0.000,B 0.000,C 90.000,E1 310.782} C_DIS
LIN {X 0.262,Y -390.610,Z 1494.495,A 0.000,B 0.000,C 90.000,E1 305.025} C_DIS
LIN {X 0.106,Y -391.104,Z 1494.493,A 0.000,B 0.000,C 90.000,E1 304.692} C_DIS
LIN {X 0.022,Y -391.648,Z 1494.489,A 0.000,B 0.000,C 90.000,E1 303.992} C_DIS
LIN {X -0.080,Y -396.825,Z 1494.459,A 0.000,B 0.000,C 90.000,E1 298.693} C_DIS
LIN {X -0.210,Y -397.120,Z 1494.457,A 0.000,B 0.000,C 90.000,E1 298.359} C_DIS
LIN {X -0.055,Y -401.597,Z 1494.426,A 0.000,B 0.000,C 90.000,E1 292.717} C_DIS
LIN {X 0.222,Y -404.659,Z 1494.395,A 0.000,B 0.000,C 90.000,E1 287.094} C_DIS
LIN {X -0.079,Y -404.735,Z 1494.391,A 0.000,B 0.000,C 90.000,E1 286.441} C_DIS
LIN {X 0.214,Y -406.099,Z 1494.364,A 0.000,B 0.000,C 90.000,E1 281.535} C_DIS
LIN {X -0.176,Y -406.094,Z 1494.362,A 0.000,B 0.000,C 90.000,E1 281.243} C_DIS
LIN {X -0.097,Y -405.680,Z 1494.333,A 0.000,B 0.000,C 90.000,E1 276.024} C_DIS
LIN {X -0.165,Y -405.058,Z 1494.328,A 0.000,B 0.000,C 90.000,E1 274.992} C_DIS
LIN {X -0.060,Y -403.497,Z 1494.304,A 0.000,B 0.000,C 90.000,E1 270.802} C_DIS
LIN {X -0.092,Y -403.288,Z 1494.302,A 0.000,B 0.000,C 90.000,E1 270.458} C_DIS
LIN {X 0.091,Y -398.931,Z 1494.271,A 0.000,B 0.000,C 90.000,E1 264.837} C_DIS
LIN {X -0.040,Y -393.108,Z 1494.242,A 0.000,B 0.000,C 90.000,E1 259.567} C_DIS
LIN {X -0.079,Y -392.835,Z 1494.240,A 0.000,B 0.000,C 90.000,E1 259.218} C_DIS
LIN {X 0.034,Y -385.993,Z 1494.212,A 0.000,B 0.000,C 90.000,E1 254.212} C_DIS
LIN {X -0.026,Y -385.267,Z 1494.208,A 0.000,B 0.000,C 90.000,E1 253.504} C_DIS
LIN {X -0.004,Y -384.768,Z 1494.206,A 0.000,B 0.000,C 90.000,E1 253.142} C_DIS
LIN {X 0.221,Y -377.973,Z 1494.182,A 0.000,B 0.000,C 90.000,E1 248.773} C_DIS
LIN {X -0.044,Y -376.233,Z 1494.174,A 0.000,B 0.000,C 90.000,E1 247.358} C_DIS
LIN {X 0.057,Y -374.944,Z 1494.170,A 0.000,B 0.000,C 90.000,E1 246.613} C_DIS
LIN {X -0.208,Y -368.417,Z 1494.148,A 0.000,B 0.000,C 90.000,E1 242.615} C_DIS
LIN {X 0.097,Y -366.047,Z 1494.137,A 0.000,B 0.000,C 90.000,E1 240.717} C_DIS
LIN {X 0.004,Y -359.196,Z 1494.115,A 0.000,B 0.000,C 90.000,E1 236.628} C_DIS
LIN {X 0.021,Y -355.842,Z 1494.100,A 0.000,B 0.000,C 90.000,E1 233.989} C_DIS
LIN {X -0.173,Y -348.793,Z 1494.075,A 0.000,B 0.000,C 90.000,E1 229.461} C_DIS
LIN {X -0.097,Y -346.185,Z 1494.062,A 0.000,B 0.000,C 90.000,E1 227.148} C_DIS
LIN {X -0.088,Y -345.065,Z 1494.058,A 0.000,B 0.000,C 90.000,E1 226.377} C_DIS
LIN {X 0.094,Y -338.586,Z 1494.030,A 0.000,B 0.000,C 90.000,E1 221.310} C_DIS
LIN {X 0.094,Y -336.840,Z 1494.019,A 0.000,B 0.000,C 90.000,E1 219.358} C_DIS
LIN {X 0.014,Y -330.861,Z 1493.988,A 0.000,B 0.000,C 90.000,E1 213.865} C_DIS
LIN {X 0.149,Y -329.296,Z 1493.975,A 0.000,B 0.000,C 90.000,E1 211.465} C_DIS
LIN {X -0.154,Y -324.669,Z 1493.942,A 0.000,B 0.000,C 90.000,E1 205.540} C_DIS
LIN {X 0.174,Y -323.837,Z 1493.928,A 0.000,B 0.000,C 90.000,E1 203.078} C_DIS
LIN {X -0.017,Y -321.124,Z 1493.881,A 0.000,B 0.000,C 90.000,E1 194.662} C_DIS
LIN {X 0.138,Y -320.932,Z 1493.877,A 0.000,B 0.000,C 90.000,E1 193.828} C_DIS
LIN {X -0.076,Y -321.562,Z 1493.832,A 0.000,B 0.000,C 90.000,E1 185.796} C_DIS
LIN {X -0.143,Y -324.415,Z 1493.790,A 0.000,B 0.000,C 90.000,E1 178.165} C_DIS
LIN {X -0.141,Y -325.376,Z 1493.783,A 0.000,B 0.000,C 90.000,E1 176.963} C_DIS
LIN {X -0.100,Y -329.112,Z 1493.750,A 0.000,B 0.000,C 90.000,E1 170.971} C_DIS
LIN {X 0.061,Y -334.260,Z 1493.726,A 0.000,B 0.000,C 90.000,E1 166.589} C_DIS
LIN {X 0.067,Y -335.488,Z 1493.719,A 0.000,B 0.000,C 90.000,E1 165.408} C_DIS
LIN {X 0.143,Y -340.932,Z 1493.695,A 0.000,B 0.000,C 90.000,E1 161.094} C_DIS
LIN {X -0.172,Y -342.138,Z 1493.691,A 0.000,B 0.000,C 90.000,E1 160.369} C_DIS
LIN {X -0.058,Y -347.939,Z 1493.667,A 0.000,B 0.000,C 90.000,E1 156.102} C_DIS
LIN {X -0.081,Y -354.259,Z 1493.648,A 0.000,B 0.000,C 90.000,E1 152.666} C_DIS
LIN {X -0.124,Y -361.124,Z 1493.626,A 0.000,B 0.000,C 90.000,E1 148.663} C_DIS
LIN {X -0.226,Y -520.265,Z 1493.626,A 0.000,B 0.000,C 90.000,E1 148.663} C_DIS
LIN {X -0.321,Y -523.251,Z 1493.625,A 0.000,B 0.000,C 90.000,E1 148.535} C_DIS
LIN {X 0.132,Y -525.006,Z 1493.624,A 0.000,B 0.000,C 90.000,E1 148.329} C_DIS
LIN {X 0.129,Y -527.116,Z 1493.623,A 0.000,B 0.000,C 90.000,E1 148.074} C_DIS
LIN {X -0.072,Y -529.886,Z 1493.620,A 0.000,B 0.000,C 90.000,E1 147.661} C_DIS
LIN {X -0.256,Y -532.039,Z 1493.618,A 0.000,B 0.000,C 90.000,E1 147.248} C_DIS
LIN {X 0.173,Y -533.297,Z 1493.616,A 0.000,B 0.000,C 90.000,E1 146.914} C_DIS
LIN {X -0.144,Y -535.428,Z 1493.613,A 0.000,B 0.000,C 90.000,E1 146.373} C_DIS
LIN {X -0.150,Y -537.214,Z 1493.610,A 0.000,B 0.000,C 90.000,E1 145.801} C_DIS
LIN {X 0.018,Y -540.443,Z 1493.604,A 0.000,B 0.000,C 90.000,E1 144.642} C_DIS
LIN {X 0.103,Y -543.276,Z 1493.597,A 0.000,B 0.000,C 90.000,E1 143.497} C_DIS
LIN {X -0.201,Y -545.700,Z 1493.591,A 0.000,B 0.000,C 90.000,E1 142.396} C_DIS
LIN {X -0.080,Y -547.296,Z 1493.586,A 0.000,B 0.000,C 90.000,E1 141.537} C_DIS
LIN {X -0.326,Y -549.176,Z 1493.580,A 0.000,B 0.000,C 90.000,E1 140.436} C_DIS
LIN {X -0.144,Y -551.257,Z 1493.572,A 0.000,B 0.000,C 90.000,E1 139.013} C_DIS
LIN {X 0.015,Y -552.729,Z 1493.566,A 0.000,B 0.000,C 90.000,E1 137.877} C_DIS
LIN {X 0.163,Y -554.057,Z 1493.560,A 0.000,B 0.000,C 90.000,E1 136.743} C_DIS
LIN {X -0.045,Y -555.263,Z 1493.554,A 0.000,B 0.000,C 90.000,E1 135.648} C_DIS
LIN {X -0.294,Y -556.077,Z 1493.549,A 0.000,B 0.000,C 90.000,E1 134.838} C_DIS
LIN {X -0.028,Y -557.295,Z 1493.541,A 0.000,B 0.000,C 90.000,E1 133.419} C_DIS
LIN {X -0.080,Y -558.446,Z 1493.532,A 0.000,B 0.000,C 90.000,E1 131.757} C_DIS
LIN {X -0.155,Y -559.208,Z 1493.524,A 0.000,B 0.000,C 90.000,E1 130.378} C_DIS
LIN {X -0.239,Y -559.661,Z 1493.518,A 0.000,B 0.000,C 90.000,E1 129.277} C_DIS
LIN {X -0.220,Y -560.164,Z 1493.510,A 0.000,B 0.000,C 90.000,E1 127.890} C_DIS
LIN {X 0.159,Y -560.412,Z 1493.504,A 0.000,B 0.000,C 90.000,E1 126.744} C_DIS
LIN {X -0.147,Y -560.575,Z 1493.497,A 0.000,B 0.000,C 90.000,E1 125.391} C_DIS
LIN {X -0.090,Y -560.517,Z 1493.490,A 0.000,B 0.000,C 90.000,E1 124.278} C_DIS
LIN {X 0.053,Y -560.391,Z 1493.483,A 0.000,B 0.000,C 90.000,E1 122.880} C_DIS
LIN {X 0.225,Y -560.421,Z 1493.472,A 0.000,B 0.000,C 90.000,E1 120.924} C_DIS
LIN {X 0.039,Y -560.650,Z 1493.463,A 0.000,B 0.000,C 90.000,E1 119.283} C_DIS
LIN {X -0.143,Y -560.882,Z 1493.453,A 0.000,B 0.000,C 90.000,E1 117.641} C_DIS
LIN {X -0.087,Y -561.154,Z 1493.444,A 0.000,B 0.000,C 90.000,E1 115.976} C_DIS
LIN {X 0.048,Y -561.588,Z 1493.434,A 0.000,B 0.000,C 90.000,E1 114.027} C_DIS
LIN {X -0.240,Y -561.908,Z 1493.427,A 0.000,B 0.000,C 90.000,E1 112.950} C_DIS
LIN {X 0.203,Y -562.310,Z 1493.417,A 0.000,B 0.000,C 90.000,E1 110.972} C_DIS
LIN {X 0.131,Y -562.705,Z 1493.407,A 0.000,B 0.000,C 90.000,E1 109.322} C_DIS
LIN {X -0.119,Y -563.141,Z 1493.398,A 0.000,B 0.000,C 90.000,E1 107.692} C_DIS
LIN {X 0.014,Y -563.571,Z 1493.389,A 0.000,B 0.000,C 90.000,E1 106.024} C_DIS
LIN {X -0.069,Y -564.257,Z 1493.377,A 0.000,B 0.000,C 90.000,E1 103.828} C_DIS
LIN {X -0.062,Y -564.807,Z 1493.368,A 0.000,B 0.000,C 90.000,E1 102.175} C_DIS
LIN {X -0.110,Y -565.573,Z 1493.357,A 0.000,B 0.000,C 90.000,E1 100.254} C_DIS
LIN {X 0.084,Y -566.231,Z 1493.349,A 0.000,B 0.000,C 90.000,E1 98.859} C_DIS
LIN {X 0.080,Y -567.199,Z 1493.337,A 0.000,B 0.000,C 90.000,E1 96.663} C_DIS
LIN {X -0.236,Y -568.131,Z 1493.328,A 0.000,B 0.000,C 90.000,E1 95.049} C_DIS
LIN {X 0.259,Y -569.481,Z 1493.316,A 0.000,B 0.000,C 90.000,E1 92.808} C_DIS
LIN {X 0.034,Y -570.703,Z 1493.305,A 0.000,B 0.000,C 90.000,E1 90.917} C_DIS
LIN {X 0.131,Y -571.658,Z 1493.298,A 0.000,B 0.000,C 90.000,E1 89.542} C_DIS
LIN {X -0.037,Y -572.987,Z 1493.287,A 0.000,B 0.000,C 90.000,E1 87.650} C_DIS
LIN {X -0.144,Y -574.249,Z 1493.276,A 0.000,B 0.000,C 90.000,E1 85.755} C_DIS
LIN {X 0.202,Y -575.355,Z 1493.267,A 0.000,B 0.000,C 90.000,E1 84.090} C_DIS
LIN {X -0.084,Y -576.306,Z 1493.260,A 0.000,B 0.000,C 90.000,E1 82.761} C_DIS
LIN {X 0.219,Y -577.351,Z 1493.252,A 0.000,B 0.000,C 90.000,E1 81.376} C_DIS
LIN {X -0.077,Y -578.846,Z 1493.242,A 0.000,B 0.000,C 90.000,E1 79.511} C_DIS
LIN {X 0.006,Y -580.156,Z 1493.233,A 0.000,B 0.000,C 90.000,E1 77.881} C_DIS
LIN {X -0.203,Y -581.445,Z 1493.224,A 0.000,B 0.000,C 90.000,E1 76.284} C_DIS
LIN {X -0.191,Y -582.399,Z 1493.216,A 0.000,B 0.000,C 90.000,E1 74.936} C_DIS
LIN {X 0.134,Y -583.268,Z 1493.209,A 0.000,B 0.000,C 90.000,E1 73.559} C_DIS
LIN {X -0.075,Y -584.040,Z 1493.201,A 0.000,B 0.000,C 90.000,E1 72.236} C_DIS
LIN {X 0.064,Y -584.646,Z 1493.195,A 0.000,B 0.000,C 90.000,E1 71.148} C_DIS
LIN {X 0.146,Y -585.647,Z 1493.185,A 0.000,B 0.000,C 90.000,E1 69.263} C_DIS
LIN {X 0.328,Y -586.886,Z 1493.173,A 0.000,B 0.000,C 90.000,E1 67.102} C_DIS
LIN {X -0.075,Y -587.856,Z 1493.164,A 0.000,B 0.000,C 90.000,E1 65.537} C_DIS
LIN {X 0.206,Y -589.001,Z 1493.154,A 0.000,B 0.000,C 90.000,E1 63.640} C_DIS
LIN {X -0.336,Y -589.892,Z 1493.146,A 0.000,B 0.000,C 90.000,E1 62.359} C_DIS
LIN {X -0.074,Y -590.838,Z 1493.139,A 0.000,B 0.000,C 90.000,E1 61.001} C_DIS
LIN {X -0.146,Y -592.653,Z 1493.126,A 0.000,B 0.000,C 90.000,E1 58.614} C_DIS
LIN {X -0.140,Y -594.101,Z 1493.115,A 0.000,B 0.000,C 90.000,E1 56.755} C_DIS
LIN {X -0.314,Y -595.414,Z 1493.106,A 0.000,B 0.000,C 90.000,E1 55.182} C_DIS
LIN {X -0.134,Y -596.493,Z 1493.098,A 0.000,B 0.000,C 90.000,E1 53.577} C_DIS
LIN {X -0.293,Y -597.161,Z 1493.090,A 0.000,B 0.000,C 90.000,E1 52.271} C_DIS
LIN {X -0.207,Y -598.117,Z 1493.079,A 0.000,B 0.000,C 90.000,E1 50.150} C_DIS
LIN {X 0.028,Y -598.552,Z 1493.074,A 0.000,B 0.000,C 90.000,E1 49.337} C_DIS
LIN {X 0.220,Y -598.854,Z 1493.067,A 0.000,B 0.000,C 90.000,E1 48.000} C_DIS
LIN {X 0.015,Y -598.911,Z 1493.063,A 0.000,B 0.000,C 90.000,E1 47.229} C_DIS
LIN {X -0.194,Y -598.852,Z 1493.058,A 0.000,B 0.000,C 90.000,E1 46.458} C_DIS
LIN {X 0.007,Y -598.608,Z 1493.051,A 0.000,B 0.000,C 90.000,E1 45.121} C_DIS
LIN {X -0.213,Y -598.300,Z 1493.046,A 0.000,B 0.000,C 90.000,E1 44.352} C_DIS
LIN {X -0.233,Y -597.686,Z 1493.041,A 0.000,B 0.000,C 90.000,E1 43.299} C_DIS
LIN {X -0.056,Y -596.609,Z 1493.033,A 0.000,B 0.000,C 90.000,E1 41.962} C_DIS
LIN {X 0.151,Y -595.284,Z 1493.026,A 0.000,B 0.000,C 90.000,E1 40.620} C_DIS
LIN {X -0.095,Y -594.269,Z 1493.021,A 0.000,B 0.000,C 90.000,E1 39.850} C_DIS
LIN {X 0.317,Y -592.754,Z 1493.016,A 0.000,B 0.000,C 90.000,E1 38.749} C_DIS
LIN {X 0.131,Y -591.464,Z 1493.011,A 0.000,B 0.000,C 90.000,E1 37.971} C_DIS
LIN {X -0.321,Y -589.461,Z 1493.005,A 0.000,B 0.000,C 90.000,E1 36.950} C_DIS
LIN {X 0.291,Y -587.782,Z 1493.001,A 0.000,B 0.000,C 90.000,E1 36.091} C_DIS
LIN {X 0.061,Y -585.859,Z 1492.996,A 0.000,B 0.000,C 90.000,E1 35.311} C_DIS
LIN {X -0.188,Y -583.688,Z 1492.992,A 0.000,B 0.000,C 90.000,E1 34.532} C_DIS
LIN {X 0.018,Y -581.333,Z 1492.987,A 0.000,B 0.000,C 90.000,E1 33.706} C_DIS
LIN {X 0.199,Y -578.556,Z 1492.983,A 0.000,B 0.000,C 90.000,E1 32.880} C_DIS
LIN {X 0.198,Y -576.513,Z 1492.980,A 0.000,B 0.000,C 90.000,E1 32.339} C_DIS
LIN {X 0.021,Y -573.079,Z 1492.975,A 0.000,B 0.000,C 90.000,E1 31.544} C_DIS
LIN {X -0.102,Y -569.935,Z 1492.972,A 0.000,B 0.000,C 90.000,E1 30.875} C_DIS
LIN {X -0.073,Y -567.709,Z 1492.969,A 0.000,B 0.000,C 90.000,E1 30.463} C_DIS
LIN {X -0.062,Y -565.111,Z 1492.967,A 0.000,B 0.000,C 90.000,E1 30.050} C_DIS
LIN {X 0.145,Y -562.019,Z 1492.965,A 0.000,B 0.000,C 90.000,E1 29.617} C_DIS
LIN {X 0.225,Y -559.404,Z 1492.963,A 0.000,B 0.000,C 90.000,E1 29.333} C_DIS
LIN {X 0.194,Y -557.849,Z 1492.962,A 0.000,B 0.000,C 90.000,E1 29.205} C_DIS
LIN {X 0.164,Y -555.712,Z 1492.962,A 0.000,B 0.000,C 90.000,E1 29.077} C_DIS
LIN {X -0.305,Y -554.053,Z 1492.961,A 0.000,B 0.000,C 90.000,E1 29.077} C_DIS
LIN {X 0.095,Y -388.668,Z 1492.961,A 0.000,B 0.000,C 90.000,E1 29.027} C_DIS
LIN {X 0.026,Y -383.025,Z 1492.939,A 0.000,B 0.000,C 90.000,E1 24.951} C_DIS
LIN {X -0.168,Y -381.310,Z 1492.933,A 0.000,B 0.000,C 90.000,E1 23.898} C_DIS
LIN {X 0.065,Y -375.141,Z 1492.906,A 0.000,B 0.000,C 90.000,E1 19.141} C_DIS
LIN {X -0.048,Y -373.415,Z 1492.896,A 0.000,B 0.000,C 90.000,E1 17.330} C_DIS
LIN {X -0.037,Y -367.898,Z 1492.868,A 0.000,B 0.000,C 90.000,E1 12.175} C_DIS
LIN {X -0.094,Y -366.498,Z 1492.855,A 0.000,B 0.000,C 90.000,E1 9.962} C_DIS
LIN {X -0.159,Y -361.799,Z 1492.822,A 0.000,B 0.000,C 90.000,E1 4.012} C_DIS
LIN {X 0.087,Y -360.903,Z 1492.801,A 0.000,B 0.000,C 90.000,E1 0.229} C_DIS
LIN {X -0.053,Y -359.426,Z 1492.770,A 0.000,B 0.000,C 90.000,E1 354.546} C_DIS
LIN {X 0.070,Y -358.890,Z 1492.759,A 0.000,B 0.000,C 90.000,E1 352.648} C_DIS
LIN {X -0.020,Y -359.563,Z 1492.726,A 0.000,B 0.000,C 90.000,E1 346.645} C_DIS
LIN {X 0.001,Y -361.801,Z 1492.684,A 0.000,B 0.000,C 90.000,E1 339.135} C_DIS
LIN {X -0.154,Y -362.053,Z 1492.680,A 0.000,B 0.000,C 90.000,E1 338.411} C_DIS
LIN {X 0.189,Y -365.980,Z 1492.643,A 0.000,B 0.000,C 90.000,E1 331.641} C_DIS
LIN {X 0.029,Y -366.387,Z 1492.639,A 0.000,B 0.000,C 90.000,E1 330.923} C_DIS
LIN {X -0.031,Y -371.355,Z 1492.604,A 0.000,B 0.000,C 90.000,E1 324.642} C_DIS
LIN {X -0.043,Y -371.766,Z 1492.602,A 0.000,B 0.000,C 90.000,E1 324.276} C_DIS
LIN {X 0.013,Y -377.358,Z 1492.567,A 0.000,B 0.000,C 90.000,E1 318.038} C_DIS
LIN {X 0.012,Y -378.235,Z 1492.563,A 0.000,B 0.000,C 90.000,E1 317.310} C_DIS
LIN {X 0.002,Y -383.940,Z 1492.531,A 0.000,B 0.000,C 90.000,E1 311.515} C_DIS
LIN {X 0.088,Y -384.893,Z 1492.527,A 0.000,B 0.000,C 90.000,E1 310.782} C_DIS
LIN {X 0.262,Y -390.610,Z 1492.495,A 0.000,B 0.000,C 90.000,E1 305.025} C_DIS
LIN {X 0.106,Y -391.104,Z 1492.493,A 0.000,B 0.000,C 90.000,E1 304.692} C_DIS
LIN {X 0.022,Y -391.648,Z 1492.489,A 0.000,B 0.000,C 90.000,E1 303.992} C_DIS
LIN {X -0.080,Y -396.825,Z 1492.459,A 0.000,B 0.000,C 90.000,E1 298.693} C_DIS
LIN {X -0.210,Y -397.120,Z 1492.457,A 0.000,B 0.000,C 90.000,E1 298.359} C_DIS
LIN {X -0.055,Y -401.597,Z 1492.426,A 0.000,B 0.000,C 90.000,E1 292.717} C_DIS
LIN {X 0.222,Y -404.659,Z 1492.395,A 0.000,B 0.000,C 90.000,E1 287.094} C_DIS
LIN {X -0.079,Y -404.735,Z 1492.391,A 0.000,B 0.000,C 90.000,E1 286.441} C_DIS
LIN {X 0.214,Y -406.099,Z 1492.364,A 0.000,B 0.000,C 90.000,E1 281.535} C_DIS
LIN {X -0.176,Y -406.094,Z 1492.362,A 0.000,B 0.000,C 90.000,E1 281.243} C_DIS
LIN {X -0.097,Y -405.680,Z 1492.333,A 0.000,B 0.000,C 90.000,E1 276.024} C_DIS
LIN {X -0.165,Y -405.058,Z 1492.328,A 0.000,B 0.000,C 90.000,E1 274.992} C_DIS
LIN {X -0.060,Y -403.497,Z 1492.304,A 0.000,B 0.000,C 90.000,E1 270.802} C_DIS
LIN {X -0.092,Y -403.288,Z 1492.302,A 0.000,B 0.000,C 90.000,E1 270.458} C_DIS
LIN {X 0.091,Y -398.931,Z 1492.271,A 0.000,B 0.000,C 90.000,E1 264.837} C_DIS
LIN {X -0.040,Y -393.108,Z 1492.242,A 0.000,B 0.000,C 90.000,E1 259.567} C_DIS
LIN {X -0.079,Y -392.835,Z 1492.240,A 0.000,B 0.000,C 90.000,E1 259.218} C_DIS
LIN {X 0.034,Y -385.993,Z 1492.212,A 0.000,B 0.000,C 90.000,E1 254.212} C_DIS
LIN {X -0.026,Y -385.267,Z 1492.208,A 0.000,B 0.000,C 90.000,E1 253.504} C_DIS
LIN {X -0.004,Y -384.768,Z 1492.206,A 0.000,B 0.000,C 90.000,E1 253.142} C_DIS
LIN {X 0.221,Y -377.973,Z 1492.182,A 0.000,B 0.000,C 90.000,E1 248.773} C_DIS
LIN {X -0.044,Y -376.233,Z 1492.174,A 0.000,B 0.000,C 90.000,E1 247.358} C_DIS
LIN {X 0.057,Y -374.944,Z 1492.170,A 0.000,B 0.000,C 90.000,E1 246.613} C_DIS
LIN {X -0.208,Y -368.417,Z 1492.148,A 0.000,B 0.000,C 90.000,E1 242.615} C_DIS
LIN {X 0.097,Y -366.047,Z 1492.137,A 0.000,B 0.000,C 90.000,E1 240.717} C_DIS
LIN {X 0.004,Y -359.196,Z 1492.115,A 0.000,B 0.000,C 90.000,E1 236.628} C_DIS
LIN {X 0.021,Y -355.842,Z 1492.100,A 0.000,B 0.000,C 90.000,E1 233.989} C_DIS
LIN {X -0.173,Y -348.793,Z 1492.075,A 0.000,B 0.000,C 90.000,E1 229.461} C_DIS
LIN {X -0.097,Y -346.185,Z 1492.062,A 0.000,B 0.000,C 90.000,E1 227.148} C_DIS
LIN {X -0.088,Y -345.065,Z 1492.058,A 0.000,B 0.000,C 90.000,E1 226.377} C_DIS
LIN {X 0.094,Y -338.586,Z 1492.030,A 0.000,B 0.000,C 90.000,E1 221.310} C_DIS
LIN {X 0.094,Y -336.840,Z 1492.019,A 0.000,B 0.000,C 90.000,E1 219.358} C_DIS
LIN {X 0.014,Y -330.861,Z 1491.988,A 0.000,B 0.000,C 90.000,E1 213.865} C_DIS
LIN {X 0.149,Y -329.296,Z 1491.975,A 0.000,B 0.000,C 90.000,E1 211.465} C_DIS
LIN {X -0.154,Y -324.669,Z 1491.942,A 0.000,B 0.000,C 90.000,E1 205.540} C_DIS
LIN {X 0.174,Y -323.837,Z 1491.928,A 0.000,B 0.000,C 90.000,E1 203.078} C_DIS
LIN {X -0.017,Y -321.124,Z 1491.881,A 0.000,B 0.000,C 90.000,E1 194.662} C_DIS
LIN {X 0.138,Y -320.932,Z 1491.877,A 0.000,B 0.000,C 90.000,E1 193.828} C_DIS
LIN {X -0.076,Y -321.562,Z 1491.832,A 0.000,B 0.000,C 90.000,E1 185.796} C_DIS
LIN {X -0.143,Y -324.415,Z 1491.790,A 0.000,B 0.000,C 90.000,E1 178.165} C_DIS
LIN {X -0.141,Y -325.376,Z 1491.783,A 0.000,B 0.000,C 90.000,E1 176.963} C_DIS
LIN {X -0.100,Y -329.112,Z 1491.750,A 0.000,B 0.000,C 90.000,E1 170.971} C_DIS
LIN {X 0.061,Y -334.260,Z 1491.726,A 0.000,B 0.000,C 90.000,E1 166.589} C_DIS
LIN {X 0.067,Y -335.488,Z 1491.719,A 0.000,B 0.000,C 90.000,E1 165.408} C_DIS
LIN {X 0.143,Y -340.932,Z 1491.695,A 0.000,B 0.000,C 90.000,E1 161.094} C_DIS
LIN {X -0.172,Y -342.138,Z 1491.691,A 0.000,B 0.000,C 90.000,E1 160.369} C_DIS
LIN {X -0.058,Y -347.939,Z 1491.667,A 0.000,B 0.000,C 90.000,E1 156.102} C_DIS
LIN {X -0.081,Y -354.259,Z 1491.648,A 0.000,B 0.000,C 90.000,E1 152.666} C_DIS
LIN {X -0.144,Y -359.851,Z 1491.630,A 0.000,B 0.000,C 90.000,E1 149.331} C_DIS
LIN {X -0.254,Y -518.010,Z 1491.630,A 0.000,B 0.000,C 90.000,E1 149.331} C_DIS
LIN {X -0.012,Y -519.587,Z 1491.629,A 0.000,B 0.000,C 90.000,E1 149.253} C_DIS
LIN {X 0.093,Y -521.375,Z 1491.629,A 0.000,B 0.000,C 90.000,E1 149.125} C_DIS
LIN {X -0.178,Y -523.557,Z 1491.627,A 0.000,B 0.000,C 90.000,E1 148.948} C_DIS
LIN {X 0.011,Y -525.621,Z 1491.626,A 0.000,B 0.000,C 90.000,E1 148.663} C_DIS
LIN {X 0.255,Y -528.422,Z 1491.624,A 0.000,B 0.000,C 90.000,E1 148.201} C_DIS
LIN {X -0.090,Y -531.270,Z 1491.620,A 0.000,B 0.000,C 90.000,E1 147.661} C_DIS
LIN {X -0.266,Y -532.994,Z 1491.618,A 0.000,B 0.000,C 90.000,E1 147.248} C_DIS
LIN {X -0.149,Y -535.948,Z 1491.613,A 0.000,B 0.000,C 90.000,E1 146.373} C_DIS
LIN {X -0.145,Y -538.514,Z 1491.608,A 0.000,B 0.000,C 90.000,E1 145.515} C_DIS
LIN {X 0.025,Y -540.895,Z 1491.604,A 0.000,B 0.000,C 90.000,E1 144.642} C_DIS
LIN {X 0.117,Y -543.718,Z 1491.597,A 0.000,B 0.000,C 90.000,E1 143.497} C_DIS
LIN {X -0.181,Y -546.097,Z 1491.591,A 0.000,B 0.000,C 90.000,E1 142.396} C_DIS
LIN {X -0.056,Y -547.679,Z 1491.586,A 0.000,B 0.000,C 90.000,E1 141.537} C_DIS
LIN {X -0.297,Y -549.546,Z 1491.580,A 0.000,B 0.000,C 90.000,E1 140.436} C_DIS
LIN {X -0.108,Y -551.592,Z 1491.572,A 0.000,B 0.000,C 90.000,E1 139.013} C_DIS
LIN {X 0.056,Y -553.055,Z 1491.566,A 0.000,B 0.000,C 90.000,E1 137.877} C_DIS
LIN {X 0.262,Y -554.646,Z 1491.558,A 0.000,B 0.000,C 90.000,E1 136.458} C_DIS
LIN {X 0.102,Y -556.101,Z 1491.551,A 0.000,B 0.000,C 90.000,E1 135.081} C_DIS
LIN {X -0.035,Y -557.303,Z 1491.543,A 0.000,B 0.000,C 90.000,E1 133.704} C_DIS
LIN {X 0.248,Y -558.285,Z 1491.535,A 0.000,B 0.000,C 90.000,E1 132.285} C_DIS
LIN {X 0.061,Y -558.831,Z 1491.531,A 0.000,B 0.000,C 90.000,E1 131.472} C_DIS
LIN {X -0.004,Y -559.525,Z 1491.523,A 0.000,B 0.000,C 90.000,E1 130.092} C_DIS
LIN {X -0.079,Y -559.926,Z 1491.517,A 0.000,B 0.000,C 90.000,E1 128.991} C_DIS
LIN {X -0.053,Y -560.315,Z 1491.509,A 0.000,B 0.000,C 90.000,E1 127.604} C_DIS
LIN {X -0.028,Y -560.576,Z 1491.501,A 0.000,B 0.000,C 90.000,E1 126.217} C_DIS
LIN {X 0.116,Y -560.602,Z 1491.494,A 0.000,B 0.000,C 90.000,E1 124.818} C_DIS
LIN {X 0.129,Y -560.418,Z 1491.483,A 0.000,B 0.000,C 90.000,E1 122.880} C_DIS
LIN {X 0.302,Y -560.447,Z 1491.472,A 0.000,B 0.000,C 90.000,E1 120.924} C_DIS
LIN {X 0.116,Y -560.676,Z 1491.463,A 0.000,B 0.000,C 90.000,E1 119.283} C_DIS
LIN {X 0.136,Y -560.837,Z 1491.455,A 0.000,B 0.000,C 90.000,E1 117.897} C_DIS
LIN {X 0.191,Y -561.105,Z 1491.446,A 0.000,B 0.000,C 90.000,E1 116.232} C_DIS
LIN {X 0.126,Y -561.613,Z 1491.434,A 0.000,B 0.000,C 90.000,E1 114.027} C_DIS
LIN {X -0.161,Y -561.935,Z 1491.427,A 0.000,B 0.000,C 90.000,E1 112.950} C_DIS
LIN {X 0.282,Y -562.338,Z 1491.417,A 0.000,B 0.000,C 90.000,E1 110.972} C_DIS
LIN {X -0.105,Y -562.706,Z 1491.409,A 0.000,B 0.000,C 90.000,E1 109.631} C_DIS
LIN {X -0.038,Y -563.186,Z 1491.398,A 0.000,B 0.000,C 90.000,E1 107.692} C_DIS
LIN {X -0.292,Y -563.684,Z 1491.388,A 0.000,B 0.000,C 90.000,E1 105.788} C_DIS
LIN {X 0.014,Y -564.316,Z 1491.377,A 0.000,B 0.000,C 90.000,E1 103.828} C_DIS
LIN {X -0.263,Y -564.780,Z 1491.369,A 0.000,B 0.000,C 90.000,E1 102.479} C_DIS
LIN {X 0.195,Y -565.393,Z 1491.360,A 0.000,B 0.000,C 90.000,E1 100.782} C_DIS
LIN {X 0.172,Y -566.317,Z 1491.349,A 0.000,B 0.000,C 90.000,E1 98.859} C_DIS
LIN {X -0.228,Y -567.435,Z 1491.336,A 0.000,B 0.000,C 90.000,E1 96.429} C_DIS
LIN {X -0.143,Y -568.225,Z 1491.328,A 0.000,B 0.000,C 90.000,E1 95.049} C_DIS
LIN {X -0.214,Y -569.576,Z 1491.316,A 0.000,B 0.000,C 90.000,E1 92.865} C_DIS
LIN {X 0.132,Y -570.829,Z 1491.305,A 0.000,B 0.000,C 90.000,E1 90.917} C_DIS
LIN {X 0.232,Y -571.817,Z 1491.298,A 0.000,B 0.000,C 90.000,E1 89.542} C_DIS
LIN {X 0.068,Y -573.148,Z 1491.287,A 0.000,B 0.000,C 90.000,E1 87.650} C_DIS
LIN {X -0.034,Y -574.443,Z 1491.276,A 0.000,B 0.000,C 90.000,E1 85.755} C_DIS
LIN {X -0.257,Y -575.548,Z 1491.267,A 0.000,B 0.000,C 90.000,E1 84.147} C_DIS
LIN {X 0.034,Y -576.527,Z 1491.260,A 0.000,B 0.000,C 90.000,E1 82.761} C_DIS
LIN {X -0.230,Y -577.564,Z 1491.252,A 0.000,B 0.000,C 90.000,E1 81.432} C_DIS
LIN {X 0.049,Y -579.085,Z 1491.242,A 0.000,B 0.000,C 90.000,E1 79.511} C_DIS
LIN {X 0.139,Y -580.425,Z 1491.233,A 0.000,B 0.000,C 90.000,E1 77.881} C_DIS
LIN {X 0.164,Y -581.920,Z 1491.222,A 0.000,B 0.000,C 90.000,E1 75.992} C_DIS
LIN {X 0.332,Y -582.821,Z 1491.215,A 0.000,B 0.000,C 90.000,E1 74.629} C_DIS
LIN {X -0.052,Y -583.685,Z 1491.207,A 0.000,B 0.000,C 90.000,E1 73.323} C_DIS
LIN {X 0.078,Y -584.309,Z 1491.201,A 0.000,B 0.000,C 90.000,E1 72.236} C_DIS
LIN {X -0.115,Y -585.015,Z 1491.194,A 0.000,B 0.000,C 90.000,E1 70.913} C_DIS
LIN {X 0.307,Y -585.884,Z 1491.185,A 0.000,B 0.000,C 90.000,E1 69.263} C_DIS
LIN {X -0.091,Y -586.427,Z 1491.179,A 0.000,B 0.000,C 90.000,E1 68.230} C_DIS
LIN {X 0.147,Y -587.278,Z 1491.172,A 0.000,B 0.000,C 90.000,E1 66.869} C_DIS
LIN {X 0.099,Y -588.118,Z 1491.164,A 0.000,B 0.000,C 90.000,E1 65.537} C_DIS
LIN {X -0.141,Y -589.237,Z 1491.154,A 0.000,B 0.000,C 90.000,E1 63.691} C_DIS
LIN {X -0.151,Y -590.127,Z 1491.146,A 0.000,B 0.000,C 90.000,E1 62.359} C_DIS
LIN {X 0.298,Y -591.237,Z 1491.138,A 0.000,B 0.000,C 90.000,E1 60.717} C_DIS
LIN {X 0.254,Y -593.117,Z 1491.124,A 0.000,B 0.000,C 90.000,E1 58.329} C_DIS
LIN {X 0.062,Y -594.341,Z 1491.115,A 0.000,B 0.000,C 90.000,E1 56.755} C_DIS
LIN {X -0.104,Y -595.673,Z 1491.107,A 0.000,B 0.000,C 90.000,E1 55.182} C_DIS
LIN {X 0.081,Y -596.779,Z 1491.098,A 0.000,B 0.000,C 90.000,E1 53.577} C_DIS
LIN {X -0.073,Y -597.494,Z 1491.090,A 0.000,B 0.000,C 90.000,E1 52.271} C_DIS
LIN {X 0.021,Y -598.447,Z 1491.079,A 0.000,B 0.000,C 90.000,E1 50.150} C_DIS
LIN {X -0.195,Y -598.865,Z 1491.074,A 0.000,B 0.000,C 90.000,E1 49.380} C_DIS
LIN {X 0.058,Y -599.164,Z 1491.067,A 0.000,B 0.000,C 90.000,E1 48.038} C_DIS
LIN {X 0.256,Y -599.229,Z 1491.063,A 0.000,B 0.000,C 90.000,E1 47.229} C_DIS
LIN {X -0.162,Y -599.129,Z 1491.057,A 0.000,B 0.000,C 90.000,E1 46.215} C_DIS
LIN {X -0.167,Y -598.934,Z 1491.051,A 0.000,B 0.000,C 90.000,E1 45.162} C_DIS
LIN {X 0.041,Y -598.655,Z 1491.047,A 0.000,B 0.000,C 90.000,E1 44.352} C_DIS
LIN {X 0.025,Y -598.048,Z 1491.041,A 0.000,B 0.000,C 90.000,E1 43.299} C_DIS
LIN {X -0.191,Y -596.986,Z 1491.033,A 0.000,B 0.000,C 90.000,E1 42.000} C_DIS
LIN {X 0.191,Y -595.397,Z 1491.024,A 0.000,B 0.000,C 90.000,E1 40.378} C_DIS
LIN {X 0.003,Y -593.570,Z 1491.017,A 0.000,B 0.000,C 90.000,E1 39.072} C_DIS
LIN {X 0.196,Y -592.348,Z 1491.013,A 0.000,B 0.000,C 90.000,E1 38.257} C_DIS
LIN {X -0.245,Y -590.413,Z 1491.007,A 0.000,B 0.000,C 90.000,E1 37.237} C_DIS
LIN {X 0.106,Y -588.257,Z 1491.001,A 0.000,B 0.000,C 90.000,E1 36.137} C_DIS
LIN {X -0.123,Y -586.351,Z 1490.996,A 0.000,B 0.000,C 90.000,E1 35.358} C_DIS
LIN {X -0.037,Y -583.452,Z 1490.990,A 0.000,B 0.000,C 90.000,E1 34.278} C_DIS
LIN {X 0.320,Y -581.881,Z 1490.987,A 0.000,B 0.000,C 90.000,E1 33.706} C_DIS
LIN {X -0.296,Y -579.123,Z 1490.983,A 0.000,B 0.000,C 90.000,E1 32.959} C_DIS
LIN {X -0.290,Y -577.111,Z 1490.980,A 0.000,B 0.000,C 90.000,E1 32.418} C_DIS
LIN {X -0.296,Y -574.929,Z 1490.977,A 0.000,B 0.000,C 90.000,E1 31.878} C_DIS
LIN {X -0.104,Y -571.906,Z 1490.973,A 0.000,B 0.000,C 90.000,E1 31.180} C_DIS
LIN {X 0.157,Y -567.943,Z 1490.969,A 0.000,B 0.000,C 90.000,E1 30.335} C_DIS
LIN {X 0.171,Y -565.714,Z 1490.966,A 0.000,B 0.000,C 90.000,E1 29.922} C_DIS
LIN {X -0.110,Y -563.186,Z 1490.964,A 0.000,B 0.000,C 90.000,E1 29.539} C_DIS
LIN {X -0.125,Y -560.123,Z 1490.962,A 0.000,B 0.000,C 90.000,E1 29.127} C_DIS
LIN {X 0.163,Y -557.583,Z 1490.960,A 0.000,B 0.000,C 90.000,E1 28.821} C_DIS
LIN {X 0.108,Y -556.109,Z 1490.959,A 0.000,B 0.000,C 90.000,E1 28.693} C_DIS
LIN {X -0.205,Y -553.877,Z 1490.959,A 0.000,B 0.000,C 90.000,E1 28.565} C_DIS
LIN {X -0.215,Y -552.132,Z 1490.958,A 0.000,B 0.000,C 90.000,E1 28.487} C_DIS
LIN {X 0.066,Y -551.162,Z 1490.958,A 0.000,B 0.000,C 90.000,E1 28.437} C_DIS
LIN {X 0.023,Y -387.700,Z 1490.958,A 0.000,B 0.000,C 90.000,E1 28.437} C_DIS
LIN {X -0.084,Y -382.785,Z 1490.938,A 0.000,B 0.000,C 90.000,E1 24.771} C_DIS
LIN {X -0.129,Y -376.095,Z 1490.911,A 0.000,B 0.000,C 90.000,E1 20.066} C_DIS
LIN {X -0.143,Y -373.627,Z 1490.897,A 0.000,B 0.000,C 90.000,E1 17.511} C_DIS
LIN {X -0.114,Y -368.028,Z 1490.869,A 0.000,B 0.000,C 90.000,E1 12.355} C_DIS
LIN {X 0.119,Y -366.322,Z 1490.854,A 0.000,B 0.000,C 90.000,E1 9.726} C_DIS
LIN {X -0.003,Y -361.709,Z 1490.821,A 0.000,B 0.000,C 90.000,E1 3.784} C_DIS
LIN {X -0.117,Y -360.820,Z 1490.800,A 0.000,B 0.000,C 90.000,E1 0.057} C_DIS
LIN {X -0.053,Y -359.426,Z 1490.770,A 0.000,B 0.000,C 90.000,E1 354.546} C_DIS
LIN {X 0.070,Y -358.890,Z 1490.759,A 0.000,B 0.000,C 90.000,E1 352.648} C_DIS
LIN {X -0.020,Y -359.563,Z 1490.726,A 0.000,B 0.000,C 90.000,E1 346.645} C_DIS
LIN {X 0.001,Y -361.801,Z 1490.684,A 0.000,B 0.000,C 90.000,E1 339.135} C_DIS
LIN {X -0.154,Y -362.053,Z 1490.680,A 0.000,B 0.000,C 90.000,E1 338.411} C_DIS
LIN {X 0.189,Y -365.980,Z 1490.643,A 0.000,B 0.000,C 90.000,E1 331.641} C_DIS
LIN {X 0.029,Y -366.387,Z 1490.639,A 0.000,B 0.000,C 90.000,E1 330.923} C_DIS
LIN {X -0.031,Y -371.355,Z 1490.604,A 0.000,B 0.000,C 90.000,E1 324.642} C_DIS
LIN {X -0.043,Y -371.766,Z 1490.602,A 0.000,B 0.000,C 90.000,E1 324.276} C_DIS
LIN {X 0.013,Y -377.358,Z 1490.567,A 0.000,B 0.000,C 90.000,E1 318.038} C_DIS
LIN {X 0.012,Y -378.235,Z 1490.563,A 0.000,B 0.000,C 90.000,E1 317.310} C_DIS
LIN {X 0.002,Y -383.940,Z 1490.531,A 0.000,B 0.000,C 90.000,E1 311.515} C_DIS
LIN {X 0.088,Y -384.893,Z 1490.527,A 0.000,B 0.000,C 90.000,E1 310.782} C_DIS
LIN {X 0.262,Y -390.610,Z 1490.495,A 0.000,B 0.000,C 90.000,E1 305.025} C_DIS
LIN {X 0.106,Y -391.104,Z 1490.493,A 0.000,B 0.000,C 90.000,E1 304.692} C_DIS
LIN {X 0.022,Y -391.648,Z 1490.489,A 0.000,B 0.000,C 90.000,E1 303.992} C_DIS
LIN {X -0.080,Y -396.825,Z 1490.459,A 0.000,B 0.000,C 90.000,E1 298.693} C_DIS
LIN {X -0.210,Y -397.120,Z 1490.457,A 0.000,B 0.000,C 90.000,E1 298.359} C_DIS
LIN {X -0.055,Y -401.597,Z 1490.426,A 0.000,B 0.000,C 90.000,E1 292.717} C_DIS
LIN {X 0.222,Y -404.659,Z 1490.395,A 0.000,B 0.000,C 90.000,E1 287.094} C_DIS
LIN {X -0.079,Y -404.735,Z 1490.391,A 0.000,B 0.000,C 90.000,E1 286.441} C_DIS
LIN {X 0.214,Y -406.099,Z 1490.364,A 0.000,B 0.000,C 90.000,E1 281.535} C_DIS
LIN {X -0.176,Y -406.094,Z 1490.362,A 0.000,B 0.000,C 90.000,E1 281.243} C_DIS
LIN {X -0.097,Y -405.680,Z 1490.333,A 0.000,B 0.000,C 90.000,E1 276.024} C_DIS
LIN {X -0.165,Y -405.058,Z 1490.328,A 0.000,B 0.000,C 90.000,E1 274.992} C_DIS
LIN {X -0.060,Y -403.497,Z 1490.304,A 0.000,B 0.000,C 90.000,E1 270.802} C_DIS
LIN {X -0.092,Y -403.288,Z 1490.302,A 0.000,B 0.000,C 90.000,E1 270.458} C_DIS
LIN {X 0.091,Y -398.931,Z 1490.271,A 0.000,B 0.000,C 90.000,E1 264.837} C_DIS
LIN {X -0.040,Y -393.108,Z 1490.242,A 0.000,B 0.000,C 90.000,E1 259.567} C_DIS
LIN {X -0.079,Y -392.835,Z 1490.240,A 0.000,B 0.000,C 90.000,E1 259.218} C_DIS
LIN {X 0.034,Y -385.993,Z 1490.212,A 0.000,B 0.000,C 90.000,E1 254.212} C_DIS
LIN {X -0.026,Y -385.267,Z 1490.208,A 0.000,B 0.000,C 90.000,E1 253.504} C_DIS
LIN {X -0.004,Y -384.768,Z 1490.206,A 0.000,B 0.000,C 90.000,E1 253.142} C_DIS
LIN {X 0.221,Y -377.973,Z 1490.182,A 0.000,B 0.000,C 90.000,E1 248.773} C_DIS
LIN {X -0.044,Y -376.233,Z 1490.174,A 0.000,B 0.000,C 90.000,E1 247.358} C_DIS
LIN {X 0.057,Y -374.944,Z 1490.170,A 0.000,B 0.000,C 90.000,E1 246.613} C_DIS
LIN {X -0.208,Y -368.417,Z 1490.148,A 0.000,B 0.000,C 90.000,E1 242.615} C_DIS
LIN {X 0.097,Y -366.047,Z 1490.137,A 0.000,B 0.000,C 90.000,E1 240.717} C_DIS
LIN {X 0.004,Y -359.196,Z 1490.115,A 0.000,B 0.000,C 90.000,E1 236.628} C_DIS
LIN {X 0.021,Y -355.842,Z 1490.100,A 0.000,B 0.000,C 90.000,E1 233.989} C_DIS
LIN {X -0.173,Y -348.793,Z 1490.075,A 0.000,B 0.000,C 90.000,E1 229.461} C_DIS
LIN {X -0.097,Y -346.185,Z 1490.062,A 0.000,B 0.000,C 90.000,E1 227.148} C_DIS
LIN {X -0.088,Y -345.065,Z 1490.058,A 0.000,B 0.000,C 90.000,E1 226.377} C_DIS
LIN {X 0.094,Y -338.586,Z 1490.030,A 0.000,B 0.000,C 90.000,E1 221.310} C_DIS
LIN {X 0.094,Y -336.840,Z 1490.019,A 0.000,B 0.000,C 90.000,E1 219.358} C_DIS
LIN {X 0.014,Y -330.861,Z 1489.988,A 0.000,B 0.000,C 90.000,E1 213.865} C_DIS
LIN {X 0.149,Y -329.296,Z 1489.975,A 0.000,B 0.000,C 90.000,E1 211.465} C_DIS
LIN {X -0.154,Y -324.669,Z 1489.942,A 0.000,B 0.000,C 90.000,E1 205.540} C_DIS
LIN {X 0.174,Y -323.837,Z 1489.928,A 0.000,B 0.000,C 90.000,E1 203.078} C_DIS
LIN {X -0.017,Y -321.124,Z 1489.881,A 0.000,B 0.000,C 90.000,E1 194.662} C_DIS
LIN {X 0.138,Y -320.932,Z 1489.877,A 0.000,B 0.000,C 90.000,E1 193.828} C_DIS
LIN {X -0.076,Y -321.562,Z 1489.832,A 0.000,B 0.000,C 90.000,E1 185.796} C_DIS
LIN {X -0.143,Y -324.415,Z 1489.790,A 0.000,B 0.000,C 90.000,E1 178.165} C_DIS
LIN {X -0.141,Y -325.376,Z 1489.783,A 0.000,B 0.000,C 90.000,E1 176.963} C_DIS
LIN {X -0.100,Y -329.112,Z 1489.750,A 0.000,B 0.000,C 90.000,E1 170.971} C_DIS
LIN {X 0.061,Y -334.260,Z 1489.726,A 0.000,B 0.000,C 90.000,E1 166.589} C_DIS
LIN {X 0.067,Y -335.488,Z 1489.719,A 0.000,B 0.000,C 90.000,E1 165.408} C_DIS
LIN {X 0.143,Y -340.932,Z 1489.695,A 0.000,B 0.000,C 90.000,E1 161.094} C_DIS
LIN {X -0.172,Y -342.138,Z 1489.691,A 0.000,B 0.000,C 90.000,E1 160.369} C_DIS
LIN {X -0.058,Y -347.939,Z 1489.667,A 0.000,B 0.000,C 90.000,E1 156.102} C_DIS
LIN {X -0.081,Y -354.259,Z 1489.648,A 0.000,B 0.000,C 90.000,E1 152.666} C_DIS
LIN {X 0.069,Y -358.659,Z 1489.633,A 0.000,B 0.000,C 90.000,E1 149.950} C_DIS
LIN {X 0.053,Y -514.925,Z 1489.633,A 0.000,B 0.000,C 90.000,E1 149.950} C_DIS
LIN {X -0.080,Y -515.839,Z 1489.633,A 0.000,B 0.000,C 90.000,E1 149.950} C_DIS
LIN {X -0.081,Y -518.810,Z 1489.632,A 0.000,B 0.000,C 90.000,E1 149.793} C_DIS
LIN {X 0.106,Y -520.647,Z 1489.631,A 0.000,B 0.000,C 90.000,E1 149.616} C_DIS
LIN {X -0.283,Y -522.852,Z 1489.630,A 0.000,B 0.000,C 90.000,E1 149.410} C_DIS
LIN {X 0.116,Y -524.983,Z 1489.628,A 0.000,B 0.000,C 90.000,E1 149.076} C_DIS
LIN {X 0.064,Y -526.742,Z 1489.627,A 0.000,B 0.000,C 90.000,E1 148.791} C_DIS
LIN {X 0.316,Y -529.023,Z 1489.624,A 0.000,B 0.000,C 90.000,E1 148.329} C_DIS
LIN {X 0.130,Y -530.908,Z 1489.622,A 0.000,B 0.000,C 90.000,E1 147.916} C_DIS
LIN {X -0.199,Y -533.071,Z 1489.619,A 0.000,B 0.000,C 90.000,E1 147.375} C_DIS
LIN {X -0.070,Y -535.048,Z 1489.615,A 0.000,B 0.000,C 90.000,E1 146.786} C_DIS
LIN {X -0.080,Y -536.906,Z 1489.612,A 0.000,B 0.000,C 90.000,E1 146.215} C_DIS
LIN {X 0.087,Y -540.219,Z 1489.606,A 0.000,B 0.000,C 90.000,E1 145.055} C_DIS
LIN {X 0.145,Y -542.469,Z 1489.601,A 0.000,B 0.000,C 90.000,E1 144.196} C_DIS
LIN {X 0.231,Y -544.448,Z 1489.597,A 0.000,B 0.000,C 90.000,E1 143.336} C_DIS
LIN {X 0.341,Y -546.228,Z 1489.592,A 0.000,B 0.000,C 90.000,E1 142.477} C_DIS
LIN {X 0.084,Y -548.310,Z 1489.586,A 0.000,B 0.000,C 90.000,E1 141.376} C_DIS
LIN {X 0.229,Y -549.706,Z 1489.581,A 0.000,B 0.000,C 90.000,E1 140.517} C_DIS
LIN {X 0.004,Y -551.722,Z 1489.573,A 0.000,B 0.000,C 90.000,E1 139.138} C_DIS
LIN {X 0.176,Y -553.187,Z 1489.567,A 0.000,B 0.000,C 90.000,E1 138.000} C_DIS
LIN {X -0.042,Y -554.474,Z 1489.561,A 0.000,B 0.000,C 90.000,E1 136.905} C_DIS
LIN {X 0.196,Y -555.943,Z 1489.553,A 0.000,B 0.000,C 90.000,E1 135.486} C_DIS
LIN {X 0.003,Y -556.959,Z 1489.547,A 0.000,B 0.000,C 90.000,E1 134.393} C_DIS
LIN {X -0.174,Y -557.839,Z 1489.541,A 0.000,B 0.000,C 90.000,E1 133.299} C_DIS
LIN {X -0.259,Y -558.790,Z 1489.533,A 0.000,B 0.000,C 90.000,E1 131.919} C_DIS
LIN {X -0.326,Y -559.509,Z 1489.525,A 0.000,B 0.000,C 90.000,E1 130.539} C_DIS
LIN {X 0.041,Y -560.025,Z 1489.517,A 0.000,B 0.000,C 90.000,E1 129.116} C_DIS
LIN {X 0.063,Y -560.392,Z 1489.510,A 0.000,B 0.000,C 90.000,E1 127.729} C_DIS
LIN {X -0.248,Y -560.611,Z 1489.502,A 0.000,B 0.000,C 90.000,E1 126.377} C_DIS
LIN {X -0.002,Y -560.638,Z 1489.493,A 0.000,B 0.000,C 90.000,E1 124.692} C_DIS
LIN {X 0.015,Y -560.422,Z 1489.482,A 0.000,B 0.000,C 90.000,E1 122.752} C_DIS
LIN {X 0.112,Y -560.456,Z 1489.473,A 0.000,B 0.000,C 90.000,E1 121.082} C_DIS
LIN {X 0.010,Y -560.713,Z 1489.462,A 0.000,B 0.000,C 90.000,E1 119.155} C_DIS
LIN {X -0.170,Y -560.907,Z 1489.453,A 0.000,B 0.000,C 90.000,E1 117.513} C_DIS
LIN {X -0.112,Y -561.215,Z 1489.444,A 0.000,B 0.000,C 90.000,E1 115.848} C_DIS
LIN {X 0.023,Y -561.667,Z 1489.433,A 0.000,B 0.000,C 90.000,E1 113.898} C_DIS
LIN {X 0.253,Y -561.979,Z 1489.427,A 0.000,B 0.000,C 90.000,E1 112.770} C_DIS
LIN {X -0.025,Y -562.408,Z 1489.416,A 0.000,B 0.000,C 90.000,E1 110.865} C_DIS
LIN {X -0.213,Y -562.784,Z 1489.408,A 0.000,B 0.000,C 90.000,E1 109.504} C_DIS
LIN {X -0.320,Y -563.257,Z 1489.398,A 0.000,B 0.000,C 90.000,E1 107.583} C_DIS
LIN {X -0.022,Y -563.693,Z 1489.388,A 0.000,B 0.000,C 90.000,E1 105.898} C_DIS
LIN {X 0.140,Y -564.318,Z 1489.378,A 0.000,B 0.000,C 90.000,E1 103.953} C_DIS
LIN {X 0.160,Y -564.890,Z 1489.368,A 0.000,B 0.000,C 90.000,E1 102.299} C_DIS
LIN {X 0.226,Y -565.646,Z 1489.358,A 0.000,B 0.000,C 90.000,E1 100.366} C_DIS
LIN {X -0.060,Y -566.439,Z 1489.349,A 0.000,B 0.000,C 90.000,E1 98.746} C_DIS
LIN {X -0.053,Y -567.441,Z 1489.336,A 0.000,B 0.000,C 90.000,E1 96.549} C_DIS
LIN {X 0.205,Y -568.388,Z 1489.327,A 0.000,B 0.000,C 90.000,E1 94.878} C_DIS
LIN {X 0.145,Y -569.769,Z 1489.315,A 0.000,B 0.000,C 90.000,E1 92.694} C_DIS
LIN {X -0.073,Y -571.056,Z 1489.304,A 0.000,B 0.000,C 90.000,E1 90.802} C_DIS
LIN {X 0.167,Y -572.218,Z 1489.295,A 0.000,B 0.000,C 90.000,E1 89.141} C_DIS
LIN {X -0.269,Y -573.192,Z 1489.288,A 0.000,B 0.000,C 90.000,E1 87.822} C_DIS
LIN {X 0.205,Y -574.503,Z 1489.277,A 0.000,B 0.000,C 90.000,E1 85.869} C_DIS
LIN {X 0.123,Y -575.831,Z 1489.267,A 0.000,B 0.000,C 90.000,E1 83.976} C_DIS
LIN {X -0.157,Y -576.824,Z 1489.259,A 0.000,B 0.000,C 90.000,E1 82.648} C_DIS
LIN {X -0.207,Y -578.095,Z 1489.250,A 0.000,B 0.000,C 90.000,E1 81.027} C_DIS
LIN {X -0.139,Y -579.405,Z 1489.241,A 0.000,B 0.000,C 90.000,E1 79.398} C_DIS
LIN {X 0.073,Y -580.777,Z 1489.232,A 0.000,B 0.000,C 90.000,E1 77.757} C_DIS
LIN {X -0.025,Y -582.242,Z 1489.222,A 0.000,B 0.000,C 90.000,E1 75.880} C_DIS
LIN {X 0.142,Y -583.167,Z 1489.214,A 0.000,B 0.000,C 90.000,E1 74.519} C_DIS
LIN {X -0.075,Y -584.013,Z 1489.207,A 0.000,B 0.000,C 90.000,E1 73.196} C_DIS
LIN {X -0.116,Y -584.621,Z 1489.201,A 0.000,B 0.000,C 90.000,E1 72.127} C_DIS
LIN {X -0.120,Y -585.315,Z 1489.193,A 0.000,B 0.000,C 90.000,E1 70.786} C_DIS
LIN {X 0.104,Y -586.190,Z 1489.184,A 0.000,B 0.000,C 90.000,E1 69.156} C_DIS
LIN {X -0.255,Y -587.403,Z 1489.172,A 0.000,B 0.000,C 90.000,E1 67.050} C_DIS
LIN {X 0.237,Y -588.286,Z 1489.165,A 0.000,B 0.000,C 90.000,E1 65.665} C_DIS
LIN {X -0.106,Y -589.510,Z 1489.153,A 0.000,B 0.000,C 90.000,E1 63.563} C_DIS
LIN {X -0.219,Y -590.573,Z 1489.144,A 0.000,B 0.000,C 90.000,E1 61.975} C_DIS
LIN {X 0.342,Y -591.563,Z 1489.137,A 0.000,B 0.000,C 90.000,E1 60.589} C_DIS
LIN {X 0.100,Y -593.237,Z 1489.125,A 0.000,B 0.000,C 90.000,E1 58.486} C_DIS
LIN {X -0.099,Y -594.496,Z 1489.116,A 0.000,B 0.000,C 90.000,E1 56.914} C_DIS
LIN {X -0.048,Y -596.019,Z 1489.106,A 0.000,B 0.000,C 90.000,E1 55.055} C_DIS
LIN {X 0.262,Y -596.965,Z 1489.099,A 0.000,B 0.000,C 90.000,E1 53.703} C_DIS
LIN {X 0.117,Y -597.722,Z 1489.091,A 0.000,B 0.000,C 90.000,E1 52.396} C_DIS
LIN {X -0.014,Y -598.263,Z 1489.084,A 0.000,B 0.000,C 90.000,E1 51.090} C_DIS
LIN {X 0.005,Y -598.827,Z 1489.078,A 0.000,B 0.000,C 90.000,E1 50.033} C_DIS
LIN {X 0.255,Y -599.229,Z 1489.074,A 0.000,B 0.000,C 90.000,E1 49.218} C_DIS
LIN {X 0.285,Y -599.447,Z 1489.068,A 0.000,B 0.000,C 90.000,E1 48.162} C_DIS
LIN {X -0.129,Y -599.506,Z 1489.062,A 0.000,B 0.000,C 90.000,E1 47.148} C_DIS
LIN {X -0.331,Y -599.504,Z 1489.057,A 0.000,B 0.000,C 90.000,E1 46.377} C_DIS
LIN {X -0.331,Y -599.294,Z 1489.052,A 0.000,B 0.000,C 90.000,E1 45.324} C_DIS
LIN {X -0.120,Y -599.071,Z 1489.047,A 0.000,B 0.000,C 90.000,E1 44.514} C_DIS
LIN {X 0.092,Y -598.263,Z 1489.040,A 0.000,B 0.000,C 90.000,E1 43.176} C_DIS
LIN {X 0.065,Y -597.454,Z 1489.034,A 0.000,B 0.000,C 90.000,E1 42.123} C_DIS
LIN {X 0.059,Y -595.854,Z 1489.025,A 0.000,B 0.000,C 90.000,E1 40.539} C_DIS
LIN {X 0.038,Y -594.505,Z 1489.019,A 0.000,B 0.000,C 90.000,E1 39.483} C_DIS
LIN {X -0.378,Y -592.926,Z 1489.014,A 0.000,B 0.000,C 90.000,E1 38.463} C_DIS
LIN {X 0.015,Y -591.057,Z 1489.008,A 0.000,B 0.000,C 90.000,E1 37.363} C_DIS
LIN {X 0.023,Y -588.953,Z 1489.002,A 0.000,B 0.000,C 90.000,E1 36.297} C_DIS
LIN {X -0.195,Y -587.143,Z 1488.997,A 0.000,B 0.000,C 90.000,E1 35.518} C_DIS
LIN {X 0.048,Y -585.068,Z 1488.993,A 0.000,B 0.000,C 90.000,E1 34.692} C_DIS
LIN {X -0.210,Y -582.766,Z 1488.988,A 0.000,B 0.000,C 90.000,E1 33.913} C_DIS
LIN {X -0.012,Y -580.160,Z 1488.984,A 0.000,B 0.000,C 90.000,E1 33.086} C_DIS
LIN {X -0.155,Y -577.092,Z 1488.979,A 0.000,B 0.000,C 90.000,E1 32.291} C_DIS
LIN {X -0.162,Y -574.933,Z 1488.976,A 0.000,B 0.000,C 90.000,E1 31.750} C_DIS
LIN {X -0.052,Y -571.254,Z 1488.972,A 0.000,B 0.000,C 90.000,E1 30.924} C_DIS
LIN {X -0.287,Y -567.234,Z 1488.967,A 0.000,B 0.000,C 90.000,E1 30.129} C_DIS
LIN {X 0.121,Y -564.395,Z 1488.964,A 0.000,B 0.000,C 90.000,E1 29.539} C_DIS
LIN {X 0.012,Y -561.045,Z 1488.961,A 0.000,B 0.000,C 90.000,E1 28.999} C_DIS
LIN {X 0.202,Y -557.925,Z 1488.959,A 0.000,B 0.000,C 90.000,E1 28.565} C_DIS
LIN {X -0.004,Y -555.419,Z 1488.957,A 0.000,B 0.000,C 90.000,E1 28.309} C_DIS
LIN {X 0.154,Y -553.933,Z 1488.957,A 0.000,B 0.000,C 90.000,E1 28.153} C_DIS
LIN {X 0.155,Y -552.312,Z 1488.956,A 0.000,B 0.000,C 90.000,E1 28.025} C_DIS
LIN {X -0.070,Y -549.670,Z 1488.955,A 0.000,B 0.000,C 90.000,E1 27.897} C_DIS
LIN {X 0.004,Y -547.889,Z 1488.955,A 0.000,B 0.000,C 90.000,E1 27.847} C_DIS
LIN {X -0.024,Y -386.788,Z 1488.955,A 0.000,B 0.000,C 90.000,E1 27.847} C_DIS
LIN {X 0.000,Y -382.905,Z 1488.938,A 0.000,B 0.000,C 90.000,E1 24.847} C_DIS
LIN {X 0.107,Y -376.196,Z 1488.912,A 0.000,B 0.000,C 90.000,E1 20.120} C_DIS
LIN {X -0.025,Y -373.703,Z 1488.898,A 0.000,B 0.000,C 90.000,E1 17.583} C_DIS
LIN {X 0.111,Y -368.099,Z 1488.869,A 0.000,B 0.000,C 90.000,E1 12.411} C_DIS
LIN {X -0.081,Y -366.422,Z 1488.855,A 0.000,B 0.000,C 90.000,E1 9.849} C_DIS
LIN {X -0.144,Y -361.749,Z 1488.822,A 0.000,B 0.000,C 90.000,E1 3.898} C_DIS
LIN {X 0.103,Y -360.873,Z 1488.801,A 0.000,B 0.000,C 90.000,E1 0.115} C_DIS
LIN {X -0.053,Y -359.426,Z 1488.770,A 0.000,B 0.000,C 90.000,E1 354.546} C_DIS
LIN {X 0.070,Y -358.890,Z 1488.759,A 0.000,B 0.000,C 90.000,E1 352.648} C_DIS
LIN {X -0.020,Y -359.563,Z 1488.726,A 0.000,B 0.000,C 90.000,E1 346.645} C_DIS
LIN {X 0.001,Y -361.801,Z 1488.684,A 0.000,B 0.000,C 90.000,E1 339.135} C_DIS
LIN {X -0.154,Y -362.053,Z 1488.680,A 0.000,B 0.000,C 90.000,E1 338.411} C_DIS
LIN {X 0.189,Y -365.980,Z 1488.643,A 0.000,B 0.000,C 90.000,E1 331.641} C_DIS
LIN {X 0.029,Y -366.387,Z 1488.639,A 0.000,B 0.000,C 90.000,E1 330.923} C_DIS
LIN {X -0.031,Y -371.355,Z 1488.604,A 0.000,B 0.000,C 90.000,E1 324.642} C_DIS
LIN {X -0.043,Y -371.766,Z 1488.602,A 0.000,B 0.000,C 90.000,E1 324.276} C_DIS
LIN {X 0.013,Y -377.358,Z 1488.567,A 0.000,B 0.000,C 90.000,E1 318.038} C_DIS
LIN {X 0.012,Y -378.235,Z 1488.563,A 0.000,B 0.000,C 90.000,E1 317.310} C_DIS
LIN {X 0.002,Y -383.940,Z 1488.531,A 0.000,B 0.000,C 90.000,E1 311.515} C_DIS
LIN {X 0.088,Y -384.893,Z 1488.527,A 0.000,B 0.000,C 90.000,E1 310.782} C_DIS
LIN {X 0.262,Y -390.610,Z 1488.495,A 0.000,B 0.000,C 90.000,E1 305.025} C_DIS
LIN {X 0.106,Y -391.104,Z 1488.493,A 0.000,B 0.000,C 90.000,E1 304.692} C_DIS
LIN {X 0.022,Y -391.648,Z 1488.489,A 0.000,B 0.000,C 90.000,E1 303.992} C_DIS
LIN {X -0.080,Y -396.825,Z 1488.459,A 0.000,B 0.000,C 90.000,E1 298.693} C_DIS
LIN {X -0.210,Y -397.120,Z 1488.457,A 0.000,B 0.000,C 90.000,E1 298.359} C_DIS
LIN {X -0.055,Y -401.597,Z 1488.426,A 0.000,B 0.000,C 90.000,E1 292.717} C_DIS
LIN {X 0.222,Y -404.659,Z 1488.395,A 0.000,B 0.000,C 90.000,E1 287.094} C_DIS
LIN {X -0.079,Y -404.735,Z 1488.391,A 0.000,B 0.000,C 90.000,E1 286.441} C_DIS
LIN {X 0.214,Y -406.099,Z 1488.364,A 0.000,B 0.000,C 90.000,E1 281.535} C_DIS
LIN {X -0.176,Y -406.094,Z 1488.362,A 0.000,B 0.000,C 90.000,E1 281.243} C_DIS
LIN {X -0.097,Y -405.680,Z 1488.333,A 0.000,B 0.000,C 90.000,E1 276.024} C_DIS
LIN {X -0.165,Y -405.058,Z 1488.328,A 0.000,B 0.000,C 90.000,E1 274.992} C_DIS
LIN {X -0.060,Y -403.497,Z 1488.304,A 0.000,B 0.000,C 90.000,E1 270.802} C_DIS
LIN {X -0.092,Y -403.288,Z 1488.302,A 0.000,B 0.000,C 90.000,E1 270.458} C_DIS
LIN {X 0.091,Y -398.931,Z 1488.271,A 0.000,B 0.000,C 90.000,E1 264.837} C_DIS
LIN {X -0.040,Y -393.108,Z 1488.242,A 0.000,B 0.000,C 90.000,E1 259.567} C_DIS
LIN {X -0.079,Y -392.835,Z 1488.240,A 0.000,B 0.000,C 90.000,E1 259.218} C_DIS
LIN {X 0.034,Y -385.993,Z 1488.212,A 0.000,B 0.000,C 90.000,E1 254.212} C_DIS
LIN {X -0.026,Y -385.267,Z 1488.208,A 0.000,B 0.000,C 90.000,E1 253.504} C_DIS
LIN {X -0.004,Y -384.768,Z 1488.206,A 0.000,B 0.000,C 90.000,E1 253.142} C_DIS
LIN {X 0.221,Y -377.973,Z 1488.182,A 0.000,B 0.000,C 90.000,E1 248.773} C_DIS
LIN {X -0.044,Y -376.233,Z 1488.174,A 0.000,B 0.000,C 90.000,E1 247.358} C_DIS
LIN {X 0.057,Y -374.944,Z 1488.170,A 0.000,B 0.000,C 90.000,E1 246.613} C_DIS
LIN {X -0.208,Y -368.417,Z 1488.148,A 0.000,B 0.000,C 90.000,E1 242.615} C_DIS
LIN {X 0.097,Y -366.047,Z 1488.137,A 0.000,B 0.000,C 90.000,E1 240.717} C_DIS
LIN {X 0.004,Y -359.196,Z 1488.115,A 0.000,B 0.000,C 90.000,E1 236.628} C_DIS
LIN {X 0.021,Y -355.842,Z 1488.100,A 0.000,B 0.000,C 90.000,E1 233.989} C_DIS
LIN {X -0.173,Y -348.793,Z 1488.075,A 0.000,B 0.000,C 90.000,E1 229.461} C_DIS
LIN {X -0.097,Y -346.185,Z 1488.062,A 0.000,B 0.000,C 90.000,E1 227.148} C_DIS
LIN {X -0.088,Y -345.065,Z 1488.058,A 0.000,B 0.000,C 90.000,E1 226.377} C_DIS
LIN {X 0.094,Y -338.586,Z 1488.030,A 0.000,B 0.000,C 90.000,E1 221.310} C_DIS
LIN {X 0.094,Y -336.840,Z 1488.019,A 0.000,B 0.000,C 90.000,E1 219.358} C_DIS
LIN {X 0.014,Y -330.861,Z 1487.988,A 0.000,B 0.000,C 90.000,E1 213.865} C_DIS
LIN {X 0.149,Y -329.296,Z 1487.975,A 0.000,B 0.000,C 90.000,E1 211.465} C_DIS
LIN {X -0.154,Y -324.669,Z 1487.942,A 0.000,B 0.000,C 90.000,E1 205.540} C_DIS
LIN {X 0.174,Y -323.837,Z 1487.928,A 0.000,B 0.000,C 90.000,E1 203.078} C_DIS
LIN {X -0.017,Y -321.124,Z 1487.881,A 0.000,B 0.000,C 90.000,E1 194.662} C_DIS
LIN {X 0.138,Y -320.932,Z 1487.877,A 0.000,B 0.000,C 90.000,E1 193.828} C_DIS
LIN {X -0.076,Y -321.562,Z 1487.832,A 0.000,B 0.000,C 90.000,E1 185.796} C_DIS
LIN {X -0.143,Y -324.415,Z 1487.790,A 0.000,B 0.000,C 90.000,E1 178.165} C_DIS
LIN {X -0.141,Y -325.376,Z 1487.783,A 0.000,B 0.000,C 90.000,E1 176.963} C_DIS
LIN {X -0.100,Y -329.112,Z 1487.750,A 0.000,B 0.000,C 90.000,E1 170.971} C_DIS
LIN {X 0.061,Y -334.260,Z 1487.726,A 0.000,B 0.000,C 90.000,E1 166.589} C_DIS
LIN {X 0.067,Y -335.488,Z 1487.719,A 0.000,B 0.000,C 90.000,E1 165.408} C_DIS
LIN {X 0.143,Y -340.932,Z 1487.695,A 0.000,B 0.000,C 90.000,E1 161.094} C_DIS
LIN {X -0.172,Y -342.138,Z 1487.691,A 0.000,B 0.000,C 90.000,E1 160.369} C_DIS
LIN {X -0.058,Y -347.939,Z 1487.667,A 0.000,B 0.000,C 90.000,E1 156.102} C_DIS
LIN {X -0.081,Y -354.259,Z 1487.648,A 0.000,B 0.000,C 90.000,E1 152.666} C_DIS
LIN {X 0.041,Y -357.552,Z 1487.637,A 0.000,B 0.000,C 90.000,E1 150.589} C_DIS
LIN {X 0.028,Y -512.222,Z 1487.637,A 0.000,B 0.000,C 90.000,E1 150.589} C_DIS
LIN {X -0.059,Y -512.778,Z 1487.637,A 0.000,B 0.000,C 90.000,E1 150.589} C_DIS
LIN {X 0.186,Y -515.055,Z 1487.636,A 0.000,B 0.000,C 90.000,E1 150.461} C_DIS
LIN {X -0.017,Y -516.498,Z 1487.635,A 0.000,B 0.000,C 90.000,E1 150.383} C_DIS
LIN {X 0.327,Y -518.905,Z 1487.634,A 0.000,B 0.000,C 90.000,E1 150.127} C_DIS
LIN {X -0.148,Y -521.152,Z 1487.633,A 0.000,B 0.000,C 90.000,E1 149.921} C_DIS
LIN {X -0.030,Y -523.330,Z 1487.631,A 0.000,B 0.000,C 90.000,E1 149.616} C_DIS
LIN {X -0.252,Y -525.957,Z 1487.629,A 0.000,B 0.000,C 90.000,E1 149.203} C_DIS
LIN {X 0.151,Y -527.488,Z 1487.627,A 0.000,B 0.000,C 90.000,E1 148.869} C_DIS
LIN {X 0.095,Y -530.571,Z 1487.623,A 0.000,B 0.000,C 90.000,E1 148.152} C_DIS
LIN {X 0.025,Y -533.777,Z 1487.618,A 0.000,B 0.000,C 90.000,E1 147.296} C_DIS
LIN {X 0.162,Y -535.714,Z 1487.615,A 0.000,B 0.000,C 90.000,E1 146.707} C_DIS
LIN {X -0.131,Y -539.214,Z 1487.609,A 0.000,B 0.000,C 90.000,E1 145.595} C_DIS
LIN {X -0.084,Y -541.595,Z 1487.604,A 0.000,B 0.000,C 90.000,E1 144.736} C_DIS
LIN {X 0.115,Y -543.701,Z 1487.599,A 0.000,B 0.000,C 90.000,E1 143.863} C_DIS
LIN {X -0.187,Y -546.172,Z 1487.593,A 0.000,B 0.000,C 90.000,E1 142.763} C_DIS
LIN {X -0.015,Y -548.257,Z 1487.587,A 0.000,B 0.000,C 90.000,E1 141.618} C_DIS
LIN {X -0.250,Y -550.126,Z 1487.581,A 0.000,B 0.000,C 90.000,E1 140.517} C_DIS
LIN {X -0.052,Y -552.109,Z 1487.573,A 0.000,B 0.000,C 90.000,E1 139.094} C_DIS
LIN {X -0.236,Y -553.908,Z 1487.565,A 0.000,B 0.000,C 90.000,E1 137.715} C_DIS
LIN {X -0.361,Y -555.708,Z 1487.556,A 0.000,B 0.000,C 90.000,E1 136.053} C_DIS
LIN {X -0.162,Y -556.772,Z 1487.550,A 0.000,B 0.000,C 90.000,E1 134.919} C_DIS
LIN {X -0.288,Y -557.904,Z 1487.542,A 0.000,B 0.000,C 90.000,E1 133.542} C_DIS
LIN {X 0.003,Y -558.852,Z 1487.534,A 0.000,B 0.000,C 90.000,E1 132.123} C_DIS
LIN {X 0.272,Y -559.433,Z 1487.528,A 0.000,B 0.000,C 90.000,E1 130.987} C_DIS
LIN {X -0.150,Y -559.988,Z 1487.520,A 0.000,B 0.000,C 90.000,E1 129.644} C_DIS
LIN {X -0.126,Y -560.362,Z 1487.513,A 0.000,B 0.000,C 90.000,E1 128.257} C_DIS
LIN {X -0.190,Y -560.566,Z 1487.506,A 0.000,B 0.000,C 90.000,E1 127.156} C_DIS
LIN {X 0.190,Y -560.689,Z 1487.500,A 0.000,B 0.000,C 90.000,E1 126.011} C_DIS
LIN {X -0.122,Y -560.667,Z 1487.493,A 0.000,B 0.000,C 90.000,E1 124.659} C_DIS
LIN {X 0.049,Y -560.438,Z 1487.482,A 0.000,B 0.000,C 90.000,E1 122.704} C_DIS
LIN {X -0.037,Y -560.458,Z 1487.473,A 0.000,B 0.000,C 90.000,E1 121.052} C_DIS
LIN {X -0.226,Y -560.682,Z 1487.463,A 0.000,B 0.000,C 90.000,E1 119.411} C_DIS
LIN {X -0.004,Y -560.800,Z 1487.457,A 0.000,B 0.000,C 90.000,E1 118.281} C_DIS
LIN {X -0.152,Y -561.102,Z 1487.446,A 0.000,B 0.000,C 90.000,E1 116.360} C_DIS
LIN {X 0.012,Y -561.600,Z 1487.434,A 0.000,B 0.000,C 90.000,E1 114.131} C_DIS
LIN {X -0.186,Y -561.988,Z 1487.426,A 0.000,B 0.000,C 90.000,E1 112.770} C_DIS
LIN {X 0.262,Y -562.473,Z 1487.416,A 0.000,B 0.000,C 90.000,E1 110.791} C_DIS
LIN {X -0.121,Y -562.850,Z 1487.408,A 0.000,B 0.000,C 90.000,E1 109.450} C_DIS
LIN {X 0.172,Y -563.257,Z 1487.399,A 0.000,B 0.000,C 90.000,E1 107.764} C_DIS
LIN {X -0.068,Y -563.669,Z 1487.390,A 0.000,B 0.000,C 90.000,E1 106.134} C_DIS
LIN {X -0.071,Y -564.180,Z 1487.380,A 0.000,B 0.000,C 90.000,E1 104.481} C_DIS
LIN {X -0.055,Y -564.789,Z 1487.371,A 0.000,B 0.000,C 90.000,E1 102.827} C_DIS
LIN {X 0.012,Y -565.491,Z 1487.361,A 0.000,B 0.000,C 90.000,E1 100.894} C_DIS
LIN {X -0.184,Y -566.236,Z 1487.351,A 0.000,B 0.000,C 90.000,E1 99.265} C_DIS
LIN {X 0.017,Y -566.827,Z 1487.344,A 0.000,B 0.000,C 90.000,E1 97.871} C_DIS
LIN {X -0.152,Y -567.842,Z 1487.333,A 0.000,B 0.000,C 90.000,E1 95.967} C_DIS
LIN {X 0.054,Y -568.799,Z 1487.324,A 0.000,B 0.000,C 90.000,E1 94.302} C_DIS
LIN {X -0.282,Y -569.898,Z 1487.315,A 0.000,B 0.000,C 90.000,E1 92.694} C_DIS
LIN {X 0.075,Y -571.219,Z 1487.304,A 0.000,B 0.000,C 90.000,E1 90.745} C_DIS
LIN {X -0.117,Y -572.567,Z 1487.294,A 0.000,B 0.000,C 90.000,E1 88.854} C_DIS
LIN {X 0.025,Y -573.528,Z 1487.286,A 0.000,B 0.000,C 90.000,E1 87.478} C_DIS
LIN {X -0.071,Y -574.876,Z 1487.276,A 0.000,B 0.000,C 90.000,E1 85.584} C_DIS
LIN {X -0.093,Y -576.255,Z 1487.265,A 0.000,B 0.000,C 90.000,E1 83.685} C_DIS
LIN {X -0.022,Y -577.689,Z 1487.254,A 0.000,B 0.000,C 90.000,E1 81.781} C_DIS
LIN {X 0.038,Y -578.984,Z 1487.245,A 0.000,B 0.000,C 90.000,E1 80.151} C_DIS
LIN {X -0.094,Y -580.108,Z 1487.238,A 0.000,B 0.000,C 90.000,E1 78.814} C_DIS
LIN {X -0.095,Y -581.258,Z 1487.230,A 0.000,B 0.000,C 90.000,E1 77.465} C_DIS
LIN {X 0.149,Y -582.500,Z 1487.221,A 0.000,B 0.000,C 90.000,E1 75.825} C_DIS
LIN {X -0.246,Y -583.459,Z 1487.214,A 0.000,B 0.000,C 90.000,E1 74.519} C_DIS
LIN {X 0.101,Y -584.287,Z 1487.206,A 0.000,B 0.000,C 90.000,E1 73.142} C_DIS
LIN {X -0.093,Y -585.018,Z 1487.199,A 0.000,B 0.000,C 90.000,E1 71.819} C_DIS
LIN {X -0.083,Y -585.685,Z 1487.192,A 0.000,B 0.000,C 90.000,E1 70.477} C_DIS
LIN {X 0.150,Y -586.605,Z 1487.183,A 0.000,B 0.000,C 90.000,E1 68.847} C_DIS
LIN {X 0.105,Y -588.209,Z 1487.168,A 0.000,B 0.000,C 90.000,E1 66.177} C_DIS
LIN {X 0.300,Y -588.685,Z 1487.163,A 0.000,B 0.000,C 90.000,E1 65.357} C_DIS
LIN {X 0.066,Y -589.739,Z 1487.153,A 0.000,B 0.000,C 90.000,E1 63.512} C_DIS
LIN {X 0.125,Y -591.022,Z 1487.143,A 0.000,B 0.000,C 90.000,E1 61.641} C_DIS
LIN {X -0.109,Y -592.026,Z 1487.135,A 0.000,B 0.000,C 90.000,E1 60.333} C_DIS
LIN {X 0.070,Y -593.493,Z 1487.125,A 0.000,B 0.000,C 90.000,E1 58.456} C_DIS
LIN {X 0.389,Y -594.772,Z 1487.116,A 0.000,B 0.000,C 90.000,E1 56.834} C_DIS
LIN {X 0.226,Y -596.071,Z 1487.107,A 0.000,B 0.000,C 90.000,E1 55.261} C_DIS
LIN {X -0.063,Y -597.241,Z 1487.098,A 0.000,B 0.000,C 90.000,E1 53.703} C_DIS
LIN {X -0.204,Y -598.046,Z 1487.091,A 0.000,B 0.000,C 90.000,E1 52.396} C_DIS
LIN {X -0.099,Y -598.503,Z 1487.085,A 0.000,B 0.000,C 90.000,E1 51.331} C_DIS
LIN {X 0.153,Y -599.178,Z 1487.078,A 0.000,B 0.000,C 90.000,E1 49.989} C_DIS
LIN {X -0.052,Y -599.564,Z 1487.073,A 0.000,B 0.000,C 90.000,E1 49.218} C_DIS
LIN {X -0.017,Y -599.774,Z 1487.068,A 0.000,B 0.000,C 90.000,E1 48.162} C_DIS
LIN {X -0.214,Y -599.839,Z 1487.063,A 0.000,B 0.000,C 90.000,E1 47.391} C_DIS
LIN {X 0.222,Y -599.839,Z 1487.057,A 0.000,B 0.000,C 90.000,E1 46.296} C_DIS
LIN {X 0.015,Y -599.558,Z 1487.050,A 0.000,B 0.000,C 90.000,E1 45.000} C_DIS
LIN {X 0.229,Y -599.260,Z 1487.046,A 0.000,B 0.000,C 90.000,E1 44.190} C_DIS
LIN {X 0.225,Y -598.234,Z 1487.037,A 0.000,B 0.000,C 90.000,E1 42.609} C_DIS
LIN {X 0.016,Y -596.946,Z 1487.030,A 0.000,B 0.000,C 90.000,E1 41.310} C_DIS
LIN {X 0.014,Y -595.811,Z 1487.024,A 0.000,B 0.000,C 90.000,E1 40.253} C_DIS
LIN {X -0.228,Y -594.819,Z 1487.019,A 0.000,B 0.000,C 90.000,E1 39.483} C_DIS
LIN {X -0.055,Y -592.787,Z 1487.012,A 0.000,B 0.000,C 90.000,E1 38.141} C_DIS
LIN {X -0.029,Y -590.870,Z 1487.006,A 0.000,B 0.000,C 90.000,E1 37.076} C_DIS
LIN {X -0.023,Y -588.698,Z 1487.000,A 0.000,B 0.000,C 90.000,E1 36.011} C_DIS
LIN {X -0.244,Y -586.812,Z 1486.996,A 0.000,B 0.000,C 90.000,E1 35.231} C_DIS
LIN {X -0.004,Y -584.718,Z 1486.991,A 0.000,B 0.000,C 90.000,E1 34.405} C_DIS
LIN {X 0.215,Y -582.271,Z 1486.987,A 0.000,B 0.000,C 90.000,E1 33.579} C_DIS
LIN {X -0.246,Y -580.529,Z 1486.984,A 0.000,B 0.000,C 90.000,E1 33.086} C_DIS
LIN {X -0.230,Y -576.464,Z 1486.978,A 0.000,B 0.000,C 90.000,E1 32.005} C_DIS
LIN {X -0.107,Y -572.958,Z 1486.973,A 0.000,B 0.000,C 90.000,E1 31.180} C_DIS
LIN {X 0.079,Y -568.371,Z 1486.968,A 0.000,B 0.000,C 90.000,E1 30.207} C_DIS
LIN {X -0.181,Y -564.148,Z 1486.963,A 0.000,B 0.000,C 90.000,E1 29.411} C_DIS
LIN {X 0.299,Y -561.917,Z 1486.961,A 0.000,B 0.000,C 90.000,E1 28.949} C_DIS
LIN {X -0.095,Y -558.391,Z 1486.958,A 0.000,B 0.000,C 90.000,E1 28.437} C_DIS
LIN {X -0.141,Y -555.139,Z 1486.956,A 0.000,B 0.000,C 90.000,E1 28.025} C_DIS
LIN {X 0.134,Y -552.552,Z 1486.954,A 0.000,B 0.000,C 90.000,E1 27.719} C_DIS
LIN {X 0.026,Y -551.013,Z 1486.953,A 0.000,B 0.000,C 90.000,E1 27.590} C_DIS
LIN {X 0.048,Y -549.418,Z 1486.953,A 0.000,B 0.000,C 90.000,E1 27.462} C_DIS
LIN {X -0.162,Y -546.868,Z 1486.952,A 0.000,B 0.000,C 90.000,E1 27.334} C_DIS
LIN {X 0.038,Y -544.949,Z 1486.952,A 0.000,B 0.000,C 90.000,E1 27.257} C_DIS
LIN {X 0.003,Y -544.479,Z 1486.952,A 0.000,B 0.000,C 90.000,E1 27.257} C_DIS
LIN {X -0.022,Y -385.932,Z 1486.951,A 0.000,B 0.000,C 90.000,E1 27.257} C_DIS
LIN {X 0.089,Y -383.062,Z 1486.939,A 0.000,B 0.000,C 90.000,E1 24.975} C_DIS
LIN {X 0.058,Y -381.956,Z 1486.935,A 0.000,B 0.000,C 90.000,E1 24.259} C_DIS
LIN {X -0.173,Y -375.553,Z 1486.909,A 0.000,B 0.000,C 90.000,E1 19.577} C_DIS
LIN {X 0.064,Y -373.463,Z 1486.896,A 0.000,B 0.000,C 90.000,E1 17.347} C_DIS
LIN {X 0.107,Y -367.924,Z 1486.868,A 0.000,B 0.000,C 90.000,E1 12.187} C_DIS
LIN {X 0.128,Y -366.516,Z 1486.855,A 0.000,B 0.000,C 90.000,E1 9.962} C_DIS
LIN {X 0.062,Y -361.814,Z 1486.822,A 0.000,B 0.000,C 90.000,E1 4.012} C_DIS
LIN {X -0.053,Y -360.904,Z 1486.802,A 0.000,B 0.000,C 90.000,E1 0.286} C_DIS
LIN {X -0.053,Y -359.426,Z 1486.770,A 0.000,B 0.000,C 90.000,E1 354.546} C_DIS
LIN {X 0.070,Y -358.890,Z 1486.759,A 0.000,B 0.000,C 90.000,E1 352.648} C_DIS
LIN {X -0.020,Y -359.563,Z 1486.726,A 0.000,B 0.000,C 90.000,E1 346.645} C_DIS
LIN {X 0.001,Y -361.801,Z 1486.684,A 0.000,B 0.000,C 90.000,E1 339.135} C_DIS
LIN {X -0.154,Y -362.053,Z 1486.680,A 0.000,B 0.000,C 90.000,E1 338.411} C_DIS
LIN {X 0.189,Y -365.980,Z 1486.643,A 0.000,B 0.000,C 90.000,E1 331.641} C_DIS
LIN {X 0.029,Y -366.387,Z 1486.639,A 0.000,B 0.000,C 90.000,E1 330.923} C_DIS
LIN {X -0.031,Y -371.355,Z 1486.604,A 0.000,B 0.000,C 90.000,E1 324.642} C_DIS
LIN {X -0.043,Y -371.766,Z 1486.602,A 0.000,B 0.000,C 90.000,E1 324.276} C_DIS
LIN {X 0.013,Y -377.358,Z 1486.567,A 0.000,B 0.000,C 90.000,E1 318.038} C_DIS
LIN {X 0.012,Y -378.235,Z 1486.563,A 0.000,B 0.000,C 90.000,E1 317.310} C_DIS
LIN {X 0.002,Y -383.940,Z 1486.531,A 0.000,B 0.000,C 90.000,E1 311.515} C_DIS
LIN {X 0.088,Y -384.893,Z 1486.527,A 0.000,B 0.000,C 90.000,E1 310.782} C_DIS
LIN {X 0.262,Y -390.610,Z 1486.495,A 0.000,B 0.000,C 90.000,E1 305.025} C_DIS
LIN {X 0.106,Y -391.104,Z 1486.493,A 0.000,B 0.000,C 90.000,E1 304.692} C_DIS
LIN {X 0.022,Y -391.648,Z 1486.489,A 0.000,B 0.000,C 90.000,E1 303.992} C_DIS
LIN {X -0.080,Y -396.825,Z 1486.459,A 0.000,B 0.000,C 90.000,E1 298.693} C_DIS
LIN {X -0.210,Y -397.120,Z 1486.457,A 0.000,B 0.000,C 90.000,E1 298.359} C_DIS
LIN {X -0.055,Y -401.597,Z 1486.426,A 0.000,B 0.000,C 90.000,E1 292.717} C_DIS
LIN {X 0.222,Y -404.659,Z 1486.395,A 0.000,B 0.000,C 90.000,E1 287.094} C_DIS
LIN {X -0.079,Y -404.735,Z 1486.391,A 0.000,B 0.000,C 90.000,E1 286.441} C_DIS
LIN {X 0.214,Y -406.099,Z 1486.364,A 0.000,B 0.000,C 90.000,E1 281.535} C_DIS
LIN {X -0.176,Y -406.094,Z 1486.362,A 0.000,B 0.000,C 90.000,E1 281.243} C_DIS
LIN {X -0.097,Y -405.680,Z 1486.333,A 0.000,B 0.000,C 90.000,E1 276.024} C_DIS
LIN {X -0.165,Y -405.058,Z 1486.328,A 0.000,B 0.000,C 90.000,E1 274.992} C_DIS
LIN {X -0.060,Y -403.497,Z 1486.304,A 0.000,B 0.000,C 90.000,E1 270.802} C_DIS
LIN {X -0.092,Y -403.288,Z 1486.302,A 0.000,B 0.000,C 90.000,E1 270.458} C_DIS
LIN {X 0.091,Y -398.931,Z 1486.271,A 0.000,B 0.000,C 90.000,E1 264.837} C_DIS
LIN {X -0.040,Y -393.108,Z 1486.242,A 0.000,B 0.000,C 90.000,E1 259.567} C_DIS
LIN {X -0.079,Y -392.835,Z 1486.240,A 0.000,B 0.000,C 90.000,E1 259.218} C_DIS
LIN {X 0.034,Y -385.993,Z 1486.212,A 0.000,B 0.000,C 90.000,E1 254.212} C_DIS
LIN {X -0.026,Y -385.267,Z 1486.208,A 0.000,B 0.000,C 90.000,E1 253.504} C_DIS
LIN {X -0.004,Y -384.768,Z 1486.206,A 0.000,B 0.000,C 90.000,E1 253.142} C_DIS
LIN {X 0.221,Y -377.973,Z 1486.182,A 0.000,B 0.000,C 90.000,E1 248.773} C_DIS
LIN {X -0.044,Y -376.233,Z 1486.174,A 0.000,B 0.000,C 90.000,E1 247.358} C_DIS
LIN {X 0.057,Y -374.944,Z 1486.170,A 0.000,B 0.000,C 90.000,E1 246.613} C_DIS
LIN {X -0.208,Y -368.417,Z 1486.148,A 0.000,B 0.000,C 90.000,E1 242.615} C_DIS
LIN {X 0.097,Y -366.047,Z 1486.137,A 0.000,B 0.000,C 90.000,E1 240.717} C_DIS
LIN {X 0.004,Y -359.196,Z 1486.115,A 0.000,B 0.000,C 90.000,E1 236.628} C_DIS
LIN {X 0.021,Y -355.842,Z 1486.100,A 0.000,B 0.000,C 90.000,E1 233.989} C_DIS
LIN {X -0.173,Y -348.793,Z 1486.075,A 0.000,B 0.000,C 90.000,E1 229.461} C_DIS
LIN {X -0.097,Y -346.185,Z 1486.062,A 0.000,B 0.000,C 90.000,E1 227.148} C_DIS
LIN {X -0.088,Y -345.065,Z 1486.058,A 0.000,B 0.000,C 90.000,E1 226.377} C_DIS
LIN {X 0.094,Y -338.586,Z 1486.030,A 0.000,B 0.000,C 90.000,E1 221.310} C_DIS
LIN {X 0.094,Y -336.840,Z 1486.019,A 0.000,B 0.000,C 90.000,E1 219.358} C_DIS
LIN {X 0.014,Y -330.861,Z 1485.988,A 0.000,B 0.000,C 90.000,E1 213.865} C_DIS
LIN {X 0.149,Y -329.296,Z 1485.975,A 0.000,B 0.000,C 90.000,E1 211.465} C_DIS
LIN {X -0.154,Y -324.669,Z 1485.942,A 0.000,B 0.000,C 90.000,E1 205.540} C_DIS
LIN {X 0.174,Y -323.837,Z 1485.928,A 0.000,B 0.000,C 90.000,E1 203.078} C_DIS
LIN {X -0.017,Y -321.124,Z 1485.881,A 0.000,B 0.000,C 90.000,E1 194.662} C_DIS
LIN {X 0.138,Y -320.932,Z 1485.877,A 0.000,B 0.000,C 90.000,E1 193.828} C_DIS
LIN {X -0.076,Y -321.562,Z 1485.832,A 0.000,B 0.000,C 90.000,E1 185.796} C_DIS
LIN {X -0.143,Y -324.415,Z 1485.790,A 0.000,B 0.000,C 90.000,E1 178.165} C_DIS
LIN {X -0.141,Y -325.376,Z 1485.783,A 0.000,B 0.000,C 90.000,E1 176.963} C_DIS
LIN {X -0.100,Y -329.112,Z 1485.750,A 0.000,B 0.000,C 90.000,E1 170.971} C_DIS
LIN {X 0.061,Y -334.260,Z 1485.726,A 0.000,B 0.000,C 90.000,E1 166.589} C_DIS
LIN {X 0.067,Y -335.488,Z 1485.719,A 0.000,B 0.000,C 90.000,E1 165.408} C_DIS
LIN {X 0.143,Y -340.932,Z 1485.695,A 0.000,B 0.000,C 90.000,E1 161.094} C_DIS
LIN {X -0.172,Y -342.138,Z 1485.691,A 0.000,B 0.000,C 90.000,E1 160.369} C_DIS
LIN {X -0.058,Y -347.939,Z 1485.667,A 0.000,B 0.000,C 90.000,E1 156.102} C_DIS
LIN {X -0.081,Y -354.259,Z 1485.648,A 0.000,B 0.000,C 90.000,E1 152.666} C_DIS
LIN {X -0.062,Y -356.514,Z 1485.640,A 0.000,B 0.000,C 90.000,E1 151.229} C_DIS
LIN {X 0.311,Y -508.968,Z 1485.640,A 0.000,B 0.000,C 90.000,E1 151.179} C_DIS
LIN {X 0.069,Y -511.327,Z 1485.640,A 0.000,B 0.000,C 90.000,E1 151.129} C_DIS
LIN {X -0.274,Y -513.227,Z 1485.639,A 0.000,B 0.000,C 90.000,E1 151.051} C_DIS
LIN {X 0.248,Y -515.644,Z 1485.638,A 0.000,B 0.000,C 90.000,E1 150.795} C_DIS
LIN {X -0.089,Y -517.945,Z 1485.637,A 0.000,B 0.000,C 90.000,E1 150.589} C_DIS
LIN {X 0.122,Y -520.220,Z 1485.635,A 0.000,B 0.000,C 90.000,E1 150.284} C_DIS
LIN {X -0.118,Y -523.151,Z 1485.633,A 0.000,B 0.000,C 90.000,E1 149.871} C_DIS
LIN {X 0.110,Y -525.592,Z 1485.630,A 0.000,B 0.000,C 90.000,E1 149.410} C_DIS
LIN {X -0.256,Y -528.316,Z 1485.627,A 0.000,B 0.000,C 90.000,E1 148.869} C_DIS
LIN {X 0.125,Y -530.704,Z 1485.624,A 0.000,B 0.000,C 90.000,E1 148.250} C_DIS
LIN {X 0.229,Y -533.927,Z 1485.619,A 0.000,B 0.000,C 90.000,E1 147.375} C_DIS
LIN {X -0.083,Y -535.905,Z 1485.616,A 0.000,B 0.000,C 90.000,E1 146.834} C_DIS
LIN {X 0.074,Y -539.367,Z 1485.609,A 0.000,B 0.000,C 90.000,E1 145.674} C_DIS
LIN {X 0.122,Y -541.786,Z 1485.605,A 0.000,B 0.000,C 90.000,E1 144.815} C_DIS
LIN {X -0.117,Y -543.884,Z 1485.600,A 0.000,B 0.000,C 90.000,E1 143.989} C_DIS
LIN {X 0.021,Y -546.369,Z 1485.594,A 0.000,B 0.000,C 90.000,E1 142.844} C_DIS
LIN {X 0.194,Y -548.438,Z 1485.587,A 0.000,B 0.000,C 90.000,E1 141.698} C_DIS
LIN {X -0.039,Y -550.334,Z 1485.581,A 0.000,B 0.000,C 90.000,E1 140.598} C_DIS
LIN {X 0.162,Y -552.287,Z 1485.573,A 0.000,B 0.000,C 90.000,E1 139.175} C_DIS
LIN {X 0.002,Y -554.411,Z 1485.564,A 0.000,B 0.000,C 90.000,E1 137.514} C_DIS
LIN {X 0.300,Y -556.148,Z 1485.555,A 0.000,B 0.000,C 90.000,E1 135.810} C_DIS
LIN {X 0.060,Y -556.946,Z 1485.550,A 0.000,B 0.000,C 90.000,E1 135.000} C_DIS
LIN {X -0.061,Y -558.026,Z 1485.542,A 0.000,B 0.000,C 90.000,E1 133.623} C_DIS
LIN {X -0.142,Y -558.994,Z 1485.535,A 0.000,B 0.000,C 90.000,E1 132.243} C_DIS
LIN {X -0.284,Y -559.579,Z 1485.528,A 0.000,B 0.000,C 90.000,E1 131.148} C_DIS
LIN {X 0.087,Y -560.069,Z 1485.521,A 0.000,B 0.000,C 90.000,E1 129.725} C_DIS
LIN {X 0.115,Y -560.465,Z 1485.513,A 0.000,B 0.000,C 90.000,E1 128.338} C_DIS
LIN {X 0.053,Y -560.611,Z 1485.507,A 0.000,B 0.000,C 90.000,E1 127.237} C_DIS
LIN {X -0.250,Y -560.733,Z 1485.499,A 0.000,B 0.000,C 90.000,E1 125.884} C_DIS
LIN {X -0.096,Y -560.661,Z 1485.492,A 0.000,B 0.000,C 90.000,E1 124.485} C_DIS
LIN {X 0.007,Y -560.435,Z 1485.479,A 0.000,B 0.000,C 90.000,E1 122.260} C_DIS
LIN {X -0.035,Y -560.580,Z 1485.467,A 0.000,B 0.000,C 90.000,E1 120.050} C_DIS
LIN {X -0.291,Y -560.786,Z 1485.459,A 0.000,B 0.000,C 90.000,E1 118.693} C_DIS
LIN {X -0.175,Y -561.042,Z 1485.448,A 0.000,B 0.000,C 90.000,E1 116.744} C_DIS
LIN {X 0.282,Y -561.232,Z 1485.442,A 0.000,B 0.000,C 90.000,E1 115.591} C_DIS
LIN {X -0.208,Y -561.581,Z 1485.435,A 0.000,B 0.000,C 90.000,E1 114.259} C_DIS
LIN {X 0.110,Y -561.967,Z 1485.427,A 0.000,B 0.000,C 90.000,E1 112.845} C_DIS
LIN {X -0.275,Y -562.382,Z 1485.418,A 0.000,B 0.000,C 90.000,E1 111.227} C_DIS
LIN {X 0.066,Y -562.780,Z 1485.410,A 0.000,B 0.000,C 90.000,E1 109.812} C_DIS
LIN {X -0.179,Y -563.197,Z 1485.401,A 0.000,B 0.000,C 90.000,E1 108.181} C_DIS
LIN {X -0.270,Y -563.701,Z 1485.390,A 0.000,B 0.000,C 90.000,E1 106.260} C_DIS
LIN {X -0.125,Y -564.179,Z 1485.381,A 0.000,B 0.000,C 90.000,E1 104.592} C_DIS
LIN {X 0.047,Y -564.928,Z 1485.370,A 0.000,B 0.000,C 90.000,E1 102.647} C_DIS
LIN {X 0.110,Y -565.624,Z 1485.360,A 0.000,B 0.000,C 90.000,E1 100.715} C_DIS
LIN {X -0.178,Y -566.369,Z 1485.350,A 0.000,B 0.000,C 90.000,E1 99.095} C_DIS
LIN {X -0.269,Y -567.256,Z 1485.340,A 0.000,B 0.000,C 90.000,E1 97.182} C_DIS
LIN {X 0.145,Y -568.322,Z 1485.329,A 0.000,B 0.000,C 90.000,E1 95.220} C_DIS
LIN {X -0.080,Y -569.560,Z 1485.318,A 0.000,B 0.000,C 90.000,E1 93.326} C_DIS
LIN {X 0.163,Y -570.629,Z 1485.309,A 0.000,B 0.000,C 90.000,E1 91.661} C_DIS
LIN {X 0.120,Y -571.447,Z 1485.303,A 0.000,B 0.000,C 90.000,E1 90.573} C_DIS
LIN {X 0.073,Y -573.031,Z 1485.291,A 0.000,B 0.000,C 90.000,E1 88.396} C_DIS
LIN {X -0.182,Y -574.146,Z 1485.282,A 0.000,B 0.000,C 90.000,E1 86.788} C_DIS
LIN {X -0.262,Y -575.537,Z 1485.271,A 0.000,B 0.000,C 90.000,E1 84.894} C_DIS
LIN {X 0.167,Y -576.768,Z 1485.262,A 0.000,B 0.000,C 90.000,E1 83.223} C_DIS
LIN {X -0.109,Y -578.484,Z 1485.250,A 0.000,B 0.000,C 90.000,E1 81.084} C_DIS
LIN {X -0.252,Y -579.586,Z 1485.243,A 0.000,B 0.000,C 90.000,E1 79.746} C_DIS
LIN {X -0.154,Y -580.916,Z 1485.234,A 0.000,B 0.000,C 90.000,E1 78.117} C_DIS
LIN {X 0.319,Y -581.818,Z 1485.228,A 0.000,B 0.000,C 90.000,E1 76.992} C_DIS
LIN {X -0.221,Y -582.850,Z 1485.220,A 0.000,B 0.000,C 90.000,E1 75.700} C_DIS
LIN {X -0.041,Y -583.829,Z 1485.213,A 0.000,B 0.000,C 90.000,E1 74.338} C_DIS
LIN {X 0.314,Y -584.621,Z 1485.206,A 0.000,B 0.000,C 90.000,E1 72.960} C_DIS
LIN {X 0.128,Y -585.344,Z 1485.198,A 0.000,B 0.000,C 90.000,E1 71.638} C_DIS
LIN {X -0.193,Y -586.145,Z 1485.189,A 0.000,B 0.000,C 90.000,E1 70.061} C_DIS
LIN {X -0.167,Y -586.925,Z 1485.182,A 0.000,B 0.000,C 90.000,E1 68.720} C_DIS
LIN {X -0.197,Y -588.557,Z 1485.167,A 0.000,B 0.000,C 90.000,E1 66.049} C_DIS
LIN {X 0.002,Y -589.001,Z 1485.162,A 0.000,B 0.000,C 90.000,E1 65.229} C_DIS
LIN {X -0.117,Y -589.910,Z 1485.154,A 0.000,B 0.000,C 90.000,E1 63.640} C_DIS
LIN {X -0.263,Y -591.592,Z 1485.140,A 0.000,B 0.000,C 90.000,E1 61.257} C_DIS
LIN {X -0.298,Y -592.789,Z 1485.131,A 0.000,B 0.000,C 90.000,E1 59.665} C_DIS
LIN {X -0.099,Y -594.263,Z 1485.121,A 0.000,B 0.000,C 90.000,E1 57.788} C_DIS
LIN {X -0.099,Y -594.951,Z 1485.117,A 0.000,B 0.000,C 90.000,E1 56.993} C_DIS
LIN {X 0.298,Y -596.456,Z 1485.106,A 0.000,B 0.000,C 90.000,E1 55.102} C_DIS
LIN {X 0.024,Y -597.610,Z 1485.098,A 0.000,B 0.000,C 90.000,E1 53.543} C_DIS
LIN {X 0.131,Y -598.276,Z 1485.092,A 0.000,B 0.000,C 90.000,E1 52.477} C_DIS
LIN {X -0.230,Y -598.786,Z 1485.086,A 0.000,B 0.000,C 90.000,E1 51.457} C_DIS
LIN {X 0.272,Y -599.572,Z 1485.077,A 0.000,B 0.000,C 90.000,E1 49.828} C_DIS
LIN {X 0.073,Y -599.911,Z 1485.073,A 0.000,B 0.000,C 90.000,E1 49.057} C_DIS
LIN {X 0.329,Y -600.108,Z 1485.068,A 0.000,B 0.000,C 90.000,E1 48.243} C_DIS
LIN {X -0.079,Y -600.114,Z 1485.062,A 0.000,B 0.000,C 90.000,E1 47.229} C_DIS
LIN {X 0.363,Y -600.135,Z 1485.057,A 0.000,B 0.000,C 90.000,E1 46.134} C_DIS
LIN {X 0.162,Y -599.847,Z 1485.049,A 0.000,B 0.000,C 90.000,E1 44.838} C_DIS
LIN {X 0.378,Y -599.533,Z 1485.045,A 0.000,B 0.000,C 90.000,E1 44.028} C_DIS
LIN {X -0.026,Y -598.456,Z 1485.036,A 0.000,B 0.000,C 90.000,E1 42.486} C_DIS
LIN {X -0.056,Y -596.853,Z 1485.027,A 0.000,B 0.000,C 90.000,E1 40.906} C_DIS
LIN {X -0.064,Y -595.654,Z 1485.021,A 0.000,B 0.000,C 90.000,E1 39.850} C_DIS
LIN {X 0.146,Y -594.504,Z 1485.017,A 0.000,B 0.000,C 90.000,E1 39.036} C_DIS
LIN {X -0.024,Y -593.339,Z 1485.013,A 0.000,B 0.000,C 90.000,E1 38.257} C_DIS
LIN {X -0.238,Y -590.972,Z 1485.005,A 0.000,B 0.000,C 90.000,E1 36.950} C_DIS
LIN {X -0.227,Y -588.755,Z 1484.999,A 0.000,B 0.000,C 90.000,E1 35.884} C_DIS
LIN {X -0.248,Y -586.153,Z 1484.993,A 0.000,B 0.000,C 90.000,E1 34.818} C_DIS
LIN {X 0.130,Y -584.722,Z 1484.990,A 0.000,B 0.000,C 90.000,E1 34.246} C_DIS
LIN {X 0.197,Y -581.343,Z 1484.984,A 0.000,B 0.000,C 90.000,E1 33.166} C_DIS
LIN {X 0.225,Y -577.416,Z 1484.978,A 0.000,B 0.000,C 90.000,E1 32.084} C_DIS
LIN {X 0.375,Y -576.406,Z 1484.977,A 0.000,B 0.000,C 90.000,E1 31.799} C_DIS
LIN {X 0.198,Y -572.811,Z 1484.972,A 0.000,B 0.000,C 90.000,E1 31.003} C_DIS
LIN {X -0.107,Y -568.230,Z 1484.967,A 0.000,B 0.000,C 90.000,E1 30.079} C_DIS
LIN {X -0.092,Y -563.944,Z 1484.963,A 0.000,B 0.000,C 90.000,E1 29.255} C_DIS
LIN {X 0.016,Y -560.894,Z 1484.959,A 0.000,B 0.000,C 90.000,E1 28.693} C_DIS
LIN {X -0.016,Y -558.418,Z 1484.957,A 0.000,B 0.000,C 90.000,E1 28.281} C_DIS
LIN {X 0.165,Y -555.590,Z 1484.955,A 0.000,B 0.000,C 90.000,E1 27.847} C_DIS
LIN {X -0.156,Y -552.245,Z 1484.953,A 0.000,B 0.000,C 90.000,E1 27.462} C_DIS
LIN {X -0.125,Y -549.580,Z 1484.951,A 0.000,B 0.000,C 90.000,E1 27.180} C_DIS
LIN {X 0.276,Y -546.429,Z 1484.949,A 0.000,B 0.000,C 90.000,E1 26.873} C_DIS
LIN {X 0.148,Y -544.142,Z 1484.949,A 0.000,B 0.000,C 90.000,E1 26.744} C_DIS
LIN {X -0.037,Y -542.308,Z 1484.948,A 0.000,B 0.000,C 90.000,E1 26.693} C_DIS
LIN {X 0.060,Y -541.436,Z 1484.948,A 0.000,B 0.000,C 90.000,E1 26.668} C_DIS
LIN {X 0.008,Y -385.127,Z 1484.948,A 0.000,B 0.000,C 90.000,E1 26.668} C_DIS
LIN {X -0.060,Y -382.663,Z 1484.937,A 0.000,B 0.000,C 90.000,E1 24.695} C_DIS
LIN {X -0.128,Y -376.013,Z 1484.911,A 0.000,B 0.000,C 90.000,E1 19.993} C_DIS
LIN {X 0.090,Y -373.544,Z 1484.897,A 0.000,B 0.000,C 90.000,E1 17.402} C_DIS
LIN {X 0.128,Y -367.970,Z 1484.868,A 0.000,B 0.000,C 90.000,E1 12.243} C_DIS
LIN {X 0.146,Y -366.546,Z 1484.856,A 0.000,B 0.000,C 90.000,E1 10.018} C_DIS
LIN {X -0.141,Y -365.832,Z 1484.852,A 0.000,B 0.000,C 90.000,E1 9.321} C_DIS
LIN {X -0.126,Y -361.395,Z 1484.817,A 0.000,B 0.000,C 90.000,E1 2.980} C_DIS
LIN {X -0.035,Y -360.906,Z 1484.802,A 0.000,B 0.000,C 90.000,E1 0.344} C_DIS
LIN {X -0.092,Y -360.152,Z 1484.793,A 0.000,B 0.000,C 90.000,E1 358.682} C_DIS
LIN {X -0.053,Y -359.426,Z 1484.770,A 0.000,B 0.000,C 90.000,E1 354.546} C_DIS
LIN {X 0.070,Y -358.890,Z 1484.759,A 0.000,B 0.000,C 90.000,E1 352.648} C_DIS
LIN {X -0.020,Y -359.563,Z 1484.726,A 0.000,B 0.000,C 90.000,E1 346.645} C_DIS
LIN {X 0.001,Y -361.801,Z 1484.684,A 0.000,B 0.000,C 90.000,E1 339.135} C_DIS
LIN {X -0.154,Y -362.053,Z 1484.680,A 0.000,B 0.000,C 90.000,E1 338.411} C_DIS
LIN {X 0.189,Y -365.980,Z 1484.643,A 0.000,B 0.000,C 90.000,E1 331.641} C_DIS
LIN {X 0.029,Y -366.387,Z 1484.639,A 0.000,B 0.000,C 90.000,E1 330.923} C_DIS
LIN {X -0.031,Y -371.355,Z 1484.604,A 0.000,B 0.000,C 90.000,E1 324.642} C_DIS
LIN {X -0.043,Y -371.766,Z 1484.602,A 0.000,B 0.000,C 90.000,E1 324.276} C_DIS
LIN {X 0.013,Y -377.358,Z 1484.567,A 0.000,B 0.000,C 90.000,E1 318.038} C_DIS
LIN {X 0.012,Y -378.235,Z 1484.563,A 0.000,B 0.000,C 90.000,E1 317.310} C_DIS
LIN {X 0.002,Y -383.940,Z 1484.531,A 0.000,B 0.000,C 90.000,E1 311.515} C_DIS
LIN {X 0.088,Y -384.893,Z 1484.527,A 0.000,B 0.000,C 90.000,E1 310.782} C_DIS
LIN {X 0.262,Y -390.610,Z 1484.495,A 0.000,B 0.000,C 90.000,E1 305.025} C_DIS
LIN {X 0.106,Y -391.104,Z 1484.493,A 0.000,B 0.000,C 90.000,E1 304.692} C_DIS
LIN {X 0.022,Y -391.648,Z 1484.489,A 0.000,B 0.000,C 90.000,E1 303.992} C_DIS
LIN {X -0.080,Y -396.825,Z 1484.459,A 0.000,B 0.000,C 90.000,E1 298.693} C_DIS
LIN {X -0.210,Y -397.120,Z 1484.457,A 0.000,B 0.000,C 90.000,E1 298.359} C_DIS
LIN {X -0.055,Y -401.597,Z 1484.426,A 0.000,B 0.000,C 90.000,E1 292.717} C_DIS
LIN {X 0.222,Y -404.659,Z 1484.395,A 0.000,B 0.000,C 90.000,E1 287.094} C_DIS
LIN {X -0.079,Y -404.735,Z 1484.391,A 0.000,B 0.000,C 90.000,E1 286.441} C_DIS
LIN {X 0.214,Y -406.099,Z 1484.364,A 0.000,B 0.000,C 90.000,E1 281.535} C_DIS
LIN {X -0.176,Y -406.094,Z 1484.362,A 0.000,B 0.000,C 90.000,E1 281.243} C_DIS
LIN {X -0.097,Y -405.680,Z 1484.333,A 0.000,B 0.000,C 90.000,E1 276.024} C_DIS
LIN {X -0.165,Y -405.058,Z 1484.328,A 0.000,B 0.000,C 90.000,E1 274.992} C_DIS
LIN {X -0.060,Y -403.497,Z 1484.304,A 0.000,B 0.000,C 90.000,E1 270.802} C_DIS
LIN {X -0.092,Y -403.288,Z 1484.302,A 0.000,B 0.000,C 90.000,E1 270.458} C_DIS
LIN {X 0.091,Y -398.931,Z 1484.271,A 0.000,B 0.000,C 90.000,E1 264.837} C_DIS
LIN {X -0.040,Y -393.108,Z 1484.242,A 0.000,B 0.000,C 90.000,E1 259.567} C_DIS
LIN {X -0.079,Y -392.835,Z 1484.240,A 0.000,B 0.000,C 90.000,E1 259.218} C_DIS
LIN {X 0.034,Y -385.993,Z 1484.212,A 0.000,B 0.000,C 90.000,E1 254.212} C_DIS
LIN {X -0.026,Y -385.267,Z 1484.208,A 0.000,B 0.000,C 90.000,E1 253.504} C_DIS
LIN {X -0.004,Y -384.768,Z 1484.206,A 0.000,B 0.000,C 90.000,E1 253.142} C_DIS
LIN {X 0.221,Y -377.973,Z 1484.182,A 0.000,B 0.000,C 90.000,E1 248.773} C_DIS
LIN {X -0.044,Y -376.233,Z 1484.174,A 0.000,B 0.000,C 90.000,E1 247.358} C_DIS
LIN {X 0.057,Y -374.944,Z 1484.170,A 0.000,B 0.000,C 90.000,E1 246.613} C_DIS
LIN {X -0.208,Y -368.417,Z 1484.148,A 0.000,B 0.000,C 90.000,E1 242.615} C_DIS
LIN {X 0.097,Y -366.047,Z 1484.137,A 0.000,B 0.000,C 90.000,E1 240.717} C_DIS
LIN {X 0.004,Y -359.196,Z 1484.115,A 0.000,B 0.000,C 90.000,E1 236.628} C_DIS
LIN {X 0.021,Y -355.842,Z 1484.100,A 0.000,B 0.000,C 90.000,E1 233.989} C_DIS
LIN {X -0.173,Y -348.793,Z 1484.075,A 0.000,B 0.000,C 90.000,E1 229.461} C_DIS
LIN {X -0.097,Y -346.185,Z 1484.062,A 0.000,B 0.000,C 90.000,E1 227.148} C_DIS
LIN {X -0.088,Y -345.065,Z 1484.058,A 0.000,B 0.000,C 90.000,E1 226.377} C_DIS
LIN {X 0.094,Y -338.586,Z 1484.030,A 0.000,B 0.000,C 90.000,E1 221.310} C_DIS
LIN {X 0.094,Y -336.840,Z 1484.019,A 0.000,B 0.000,C 90.000,E1 219.358} C_DIS
LIN {X 0.014,Y -330.861,Z 1483.988,A 0.000,B 0.000,C 90.000,E1 213.865} C_DIS
LIN {X 0.149,Y -329.296,Z 1483.975,A 0.000,B 0.000,C 90.000,E1 211.465} C_DIS
LIN {X -0.154,Y -324.669,Z 1483.942,A 0.000,B 0.000,C 90.000,E1 205.540} C_DIS
LIN {X 0.174,Y -323.837,Z 1483.928,A 0.000,B 0.000,C 90.000,E1 203.078} C_DIS
LIN {X -0.017,Y -321.124,Z 1483.881,A 0.000,B 0.000,C 90.000,E1 194.662} C_DIS
LIN {X 0.138,Y -320.932,Z 1483.877,A 0.000,B 0.000,C 90.000,E1 193.828} C_DIS
LIN {X -0.076,Y -321.562,Z 1483.832,A 0.000,B 0.000,C 90.000,E1 185.796} C_DIS
LIN {X -0.143,Y -324.415,Z 1483.790,A 0.000,B 0.000,C 90.000,E1 178.165} C_DIS
LIN {X -0.141,Y -325.376,Z 1483.783,A 0.000,B 0.000,C 90.000,E1 176.963} C_DIS
LIN {X -0.100,Y -329.112,Z 1483.750,A 0.000,B 0.000,C 90.000,E1 170.971} C_DIS
LIN {X 0.061,Y -334.260,Z 1483.726,A 0.000,B 0.000,C 90.000,E1 166.589} C_DIS
LIN {X 0.067,Y -335.488,Z 1483.719,A 0.000,B 0.000,C 90.000,E1 165.408} C_DIS
LIN {X 0.143,Y -340.932,Z 1483.695,A 0.000,B 0.000,C 90.000,E1 161.094} C_DIS
LIN {X -0.172,Y -342.138,Z 1483.691,A 0.000,B 0.000,C 90.000,E1 160.369} C_DIS
LIN {X -0.058,Y -347.939,Z 1483.667,A 0.000,B 0.000,C 90.000,E1 156.102} C_DIS
LIN {X -0.081,Y -354.259,Z 1483.648,A 0.000,B 0.000,C 90.000,E1 152.666} C_DIS
LIN {X 0.017,Y -355.558,Z 1483.644,A 0.000,B 0.000,C 90.000,E1 151.820} C_DIS
LIN {X -0.019,Y -505.421,Z 1483.643,A 0.000,B 0.000,C 90.000,E1 151.820} C_DIS
LIN {X -0.105,Y -506.008,Z 1483.643,A 0.000,B 0.000,C 90.000,E1 151.820} C_DIS
LIN {X 0.181,Y -509.311,Z 1483.643,A 0.000,B 0.000,C 90.000,E1 151.641} C_DIS
LIN {X 0.019,Y -511.414,Z 1483.642,A 0.000,B 0.000,C 90.000,E1 151.513} C_DIS
LIN {X -0.091,Y -513.866,Z 1483.641,A 0.000,B 0.000,C 90.000,E1 151.307} C_DIS
LIN {X -0.098,Y -516.228,Z 1483.639,A 0.000,B 0.000,C 90.000,E1 151.051} C_DIS
LIN {X 0.290,Y -518.552,Z 1483.638,A 0.000,B 0.000,C 90.000,E1 150.717} C_DIS
LIN {X -0.215,Y -521.462,Z 1483.635,A 0.000,B 0.000,C 90.000,E1 150.333} C_DIS
LIN {X -0.159,Y -524.681,Z 1483.632,A 0.000,B 0.000,C 90.000,E1 149.744} C_DIS
LIN {X 0.190,Y -527.470,Z 1483.629,A 0.000,B 0.000,C 90.000,E1 149.125} C_DIS
LIN {X 0.138,Y -530.547,Z 1483.625,A 0.000,B 0.000,C 90.000,E1 148.408} C_DIS
LIN {X -0.215,Y -533.861,Z 1483.620,A 0.000,B 0.000,C 90.000,E1 147.582} C_DIS
LIN {X -0.085,Y -536.760,Z 1483.615,A 0.000,B 0.000,C 90.000,E1 146.707} C_DIS
LIN {X 0.081,Y -540.174,Z 1483.609,A 0.000,B 0.000,C 90.000,E1 145.548} C_DIS
